// TIA Portal project "传感器对中" (V15.1)

(* hardware
DEVICE "S7-1200 station_1"  S7-1200 Station
   slot 0: "Rack_0"  S7-1200 Rack  Rack  V1.0
   slot 1: "280PLC"  CPU 1214C DC/DC/DC  6ES7 214-1AG40-0XB0  V4.2
   slot 2: "DI 16x24VDC/DQ 16xRelay_1"  SM 1223 DI16/DQ16 x relay  6ES7 223-1PL32-0XB0  V2.0
   slot 3: "DI 16/DQ 16x24VDC_1"  6ES7 223-1BL32-0XB0  V2.0
   slot 4: "DI 8x24VDC_1"  6ES7 221-1BF32-0XB0  V2.0
   slot 5: "AI 4x13BIT_1"  6ES7 231-4HD32-0XB0  V2.0
DEVICE "GSD device_1"  GSD.Device.PN
   slot 0: "机架"  Rack  V1.0
   slot 0: "1-sr-qd1"  SINAMICS V90 PN V1.0  6SL3 210-5Fxxx-xxFx  V1.00
      slot 0: "SINAMICS V90 PN V1.0"  SINAMICS V90 PN V1.0
      slot 1: "PN-IO"  PN-IO
         slot 1: "端口1"  Port 1
         slot 2: "端口2"  Port 2
      slot 1: "驱动_1"  Drive
         slot 0: "模块访问点"  Module Access Point
         slot 1: "没有 PROFIsafe"  without PROFIsafe
   slot 2: "标准报文3, PZD-5/9"  Standard telegram 3, PZD-5/9
DEVICE "GSD device_2"  GSD.Device.PN
   slot 0: "机架"  Rack  V1.0
   slot 0: "2-sr-qd2"  SINAMICS V90 PN V1.0  6SL3 210-5Fxxx-xxFx  V1.00
      slot 0: "SINAMICS V90 PN V1.0"  SINAMICS V90 PN V1.0
      slot 1: "PN-IO"  PN-IO
         slot 1: "端口1"  Port 1
         slot 2: "端口2"  Port 2
      slot 1: "驱动_1"  Drive
         slot 0: "模块访问点"  Module Access Point
         slot 1: "没有 PROFIsafe"  without PROFIsafe
   slot 2: "标准报文3, PZD-5/9"  Standard telegram 3, PZD-5/9
DEVICE "GSD device_4"  GSD.Device.PN
   slot 0: "机架"  Rack  V1.0
   slot 0: "4-sr-yz2"  SINAMICS V90 PN V1.0  6SL3 210-5Fxxx-xxFx  V1.00
      slot 0: "SINAMICS V90 PN V1.0"  SINAMICS V90 PN V1.0
      slot 1: "PN-IO"  PN-IO
         slot 1: "端口1"  Port 1
         slot 2: "端口2"  Port 2
      slot 1: "驱动_1"  Drive
         slot 0: "模块访问点"  Module Access Point
         slot 1: "没有 PROFIsafe"  without PROFIsafe
   slot 2: "标准报文3, PZD-5/9"  Standard telegram 3, PZD-5/9
DEVICE "GSD device_3"  GSD.Device.PN
   slot 0: "机架"  Rack  V1.0
   slot 0: "3-sr-yz1"  SINAMICS V90 PN V1.0  6SL3 210-5Fxxx-xxFx  V1.00
      slot 0: "SINAMICS V90 PN V1.0"  SINAMICS V90 PN V1.0
      slot 1: "PN-IO"  PN-IO
         slot 1: "端口1"  Port 1
         slot 2: "端口2"  Port 2
      slot 1: "驱动_1"  Drive
         slot 0: "模块访问点"  Module Access Point
         slot 1: "没有 PROFIsafe"  without PROFIsafe
   slot 2: "标准报文3, PZD-5/9"  Standard telegram 3, PZD-5/9
*)

// ===== PLC "280PLC"  CPU 1214C DC/DC/DC =====

VAR_GLOBAL   // PLC tag table "默认变量表"
   "角度编码器1A" AT %I0.0 : Bool;
   "角度编码器1B" AT %I0.1 : Bool;
   "角度编码器1Z" AT %I0.3 : Bool;
   "角度编码器2A" AT %I0.4 : Bool;
   "角度编码器2B" AT %I0.5 : Bool;
   "角度编码器2Z" AT %I0.7 : Bool;
   "工位1在位" AT %I1.4 : Bool;
   "工位2在位" AT %I1.5 : Bool;
   "工位1卡盘顶升进到位" AT %I2.0 : Bool;
   "工位1卡盘顶升退到位" AT %I2.1 : Bool;
   "产品扶持气缸1进到位" AT %I2.2 : Bool;
   "产品扶持气缸1退到位" AT %I2.3 : Bool;
   "输出轴夹紧气缸1进到位" AT %I5.4 : Bool;
   "输出轴夹紧气缸1退到位" AT %I5.5 : Bool;
   "输出轴花键移载气缸1进到位" AT %I2.6 : Bool;
   "输出轴花键移载气缸1退到位" AT %I2.7 : Bool;
   "输入轴夹紧气动卡盘2进到位" AT %I3.0 : Bool;
   "输入轴夹紧气动卡盘2退到位" AT %I3.1 : Bool;
   "产品扶持气缸2进到位" AT %I3.2 : Bool;
   "产品扶持气缸2退到位" AT %I3.3 : Bool;
   "输出轴夹紧气缸2进到位" AT %I5.6 : Bool;
   "输出轴夹紧气缸2退到位" AT %I5.7 : Bool;
   "输出轴花键移载气缸2进到位" AT %I3.6 : Bool;
   "输出轴花键移载气缸2退到位" AT %I3.7 : Bool;
   "工位2启动" AT %I4.0 : Bool;
   "复位按钮" AT %I4.1 : Bool;
   "工位1启动" AT %I4.2 : Bool;
   "安全光栅" AT %I4.3 : Bool;
   "安全继电器急停" AT %I4.4 : Bool;
   "安全门开关" AT %I4.5 : Bool;
   "急停按钮" AT %I4.6 : Bool;
   "气源不足指示" AT %I4.7 : Bool;
   "报警1" AT %I5.0 : Bool;
   "报警2" AT %I5.1 : Bool;
   "报警3" AT %I5.2 : Bool;
   "报警4" AT %I5.3 : Bool;
   "扭矩传感器1" AT %IW144 : Int;
   "扭矩传感器2" AT %IW146 : Int;
   "输入轴移载伺服-1_归位开关" AT %I1.0 : Bool;
   "输入轴移载伺服-2_归位开关" AT %I1.3 : Bool;
   "输入轴驱动伺服-1_Drive_IN" AT %I68.0 : "PD_TEL3_IN";
   "输入轴驱动伺服-2_Drive_IN" AT %I104.0 : "PD_TEL3_IN";
   "输入轴驱动伺服-2_Drive_IN(1)" AT %I86.0 : "PD_TEL3_IN";
   "输入轴移载伺服-1_Drive_IN" AT %I122.0 : "PD_TEL3_IN";
   "输入轴移载伺服-1_LowHwLimitSwitch" AT %I0.6 : Bool;
   "输入轴移载伺服-1_HighHwLimitSwitch" AT %I0.2 : Bool;
   "输入轴移载伺服-2_LowHwLimitSwitch" AT %I1.2 : Bool;
   "输入轴移载伺服-2_HighHwLimitSwitch" AT %I1.1 : Bool;
   "编码器计数1" AT %ID1000 : DInt;
   "编码器计数2" AT %ID1004 : DInt;
   "Tag_8" AT %IW1000 : Hw_Hsc;
   "输入轴驱动伺服-1_归位开关" AT %I3.4 : Bool;
   "输入轴驱动伺服-2_归位开关" AT %I3.5 : Bool;
   "工位2卡盘顶升进到位" AT %I2.4 : Bool;
   "工位2卡盘顶升退到位" AT %I2.5 : Bool;
   "复位1" AT %Q0.0 : Bool;
   "复位2" AT %Q0.1 : Bool;
   "复位3" AT %Q0.2 : Bool;
   "复位4" AT %Q0.3 : Bool;
   "三色灯-红" AT %Q0.4 : Bool;
   "三色灯-黄" AT %Q0.5 : Bool;
   "三色灯-绿" AT %Q0.6 : Bool;
   "蜂鸣器" AT %Q0.7 : Bool;
   "输入轴夹紧气动卡盘1进" AT %Q2.0 : Bool;
   "输入轴夹紧气动卡盘1退" AT %Q2.1 : Bool;
   "产品扶持气缸1进" AT %Q2.2 : Bool;
   "产品扶持气缸1退" AT %Q2.3 : Bool;
   "输出轴夹紧气缸1进" AT %Q2.4 : Bool;
   "输出轴夹紧气缸1退" AT %Q2.5 : Bool;
   "输出轴花键移载气缸1进" AT %Q2.6 : Bool;
   "输出轴花键移载气缸1退" AT %Q2.7 : Bool;
   "输入轴夹紧气动卡盘2进" AT %Q3.0 : Bool;
   "输入轴夹紧气动卡盘2退" AT %Q3.1 : Bool;
   "产品扶持气缸2进" AT %Q3.2 : Bool;
   "产品扶持气缸2退" AT %Q3.3 : Bool;
   "输出轴夹紧气缸2进" AT %Q3.4 : Bool;
   "输出轴夹紧气缸2退" AT %Q3.5 : Bool;
   "输出轴花键移载气缸2进" AT %Q3.6 : Bool;
   "输出轴花键移载气缸2退" AT %Q3.7 : Bool;
   "工位1两色灯-红" AT %Q4.0 : Bool;
   "工位1两色灯-绿" AT %Q4.1 : Bool;
   "工位2两色灯-红" AT %Q4.2 : Bool;
   "工位2两色灯-绿" AT %Q4.3 : Bool;
   "总气阀" AT %Q4.4 : Bool;
   "工位1采集切换" AT %Q4.6 : Bool;   // True:PGI采集False:板卡采集
   "输入轴驱动伺服-1_Drive_OUT" AT %Q64.0 : "PD_TEL3_OUT";
   "输入轴驱动伺服-2_Drive_OUT" AT %Q84.0 : "PD_TEL3_OUT";
   "输入轴驱动伺服-2_Drive_OUT(1)" AT %Q74.0 : "PD_TEL3_OUT";
   "输入轴移载伺服-1_Drive_OUT" AT %Q94.0 : "PD_TEL3_OUT";
   "工位2采集切换" AT %Q4.5 : Bool;   // True:PGI采集False:板卡采集
   "工位1卡盘顶升进" AT %Q5.0 : Bool;
   "工位1卡盘顶升退" AT %Q5.1 : Bool;
   "工位2卡盘顶升进" AT %Q5.2 : Bool;
   "工位2卡盘顶升退" AT %Q5.3 : Bool;
   "System_Byte" AT %MB1 : Byte;
   "FirstScan" AT %M1.0 : Bool;
   "DiagStatusUpdate" AT %M1.1 : Bool;
   "AlwaysTRUE" AT %M1.2 : Bool;
   "AlwaysFALSE" AT %M1.3 : Bool;
   "Clock_Byte" AT %MB0 : Byte;
   "Clock_10Hz" AT %M0.0 : Bool;
   "Clock_5Hz" AT %M0.1 : Bool;
   "Clock_2.5Hz" AT %M0.2 : Bool;
   "Clock_2Hz" AT %M0.3 : Bool;
   "Clock_1.25Hz" AT %M0.4 : Bool;
   "Clock_1Hz" AT %M0.5 : Bool;
   "Clock_0.625Hz" AT %M0.6 : Bool;
   "Clock_0.5Hz" AT %M0.7 : Bool;
   "单工位1" AT %M100.0 : Bool;
   "单工位2" AT %M100.1 : Bool;
   "程序停止" AT %M100.3 : Bool;
   "光栅启用" AT %M100.2 : Bool;
   "急停拍下故障" AT %M110.0 : Bool;
   "气源不足故障" AT %M110.1 : Bool;
   "安全门打开故障" AT %M110.2 : Bool;
   "光栅触碰故障" AT %M110.3 : Bool;
   "输入轴夹紧气动卡盘1进故障" AT %M110.4 : Bool;
   "输入轴夹紧气动卡盘1退故障" AT %M110.5 : Bool;
   "产品扶持气缸1进故障" AT %M110.6 : Bool;
   "产品扶持气缸1退故障" AT %M110.7 : Bool;
   "输出轴夹紧气缸1进故障" AT %M111.0 : Bool;
   "输出轴夹紧气缸1退故障" AT %M111.1 : Bool;
   "输出轴花键移载气缸1进故障" AT %M111.2 : Bool;
   "输出轴花键移载气缸1退故障" AT %M111.3 : Bool;
   "输入轴夹紧气动卡盘2进故障" AT %M111.4 : Bool;
   "输入轴夹紧气动卡盘2退故障" AT %M111.5 : Bool;
   "产品扶持气缸2进故障" AT %M111.6 : Bool;
   "产品扶持气缸2退故障" AT %M111.7 : Bool;
   "输出轴夹紧气缸2进故障" AT %M112.0 : Bool;
   "输出轴夹紧气缸2退故障" AT %M112.1 : Bool;
   "输出轴花键移载气缸2进故障" AT %M112.2 : Bool;
   "输出轴花键移载气缸2退故障" AT %M112.3 : Bool;
   "输入轴移载伺服1退到位故障" AT %M120.0 : Bool;
   "输入轴移载伺服1进到位故障" AT %M120.1 : Bool;
   "输入轴移载伺服2退到位故障" AT %M120.2 : Bool;
   "输入轴移载伺服2进到位故障" AT %M120.3 : Bool;
   "输入轴驱动伺服-1故障" AT %M130.0 : Bool;
   "输入轴驱动伺服-2故障" AT %M130.1 : Bool;
   "输入轴移载伺服-1故障" AT %M130.2 : Bool;
   "输入轴移载伺服-2故障" AT %M130.3 : Bool;
   "复位启动" AT %M100.4 : Bool;
   "复位完成" AT %M100.5 : Bool;
   "Tag_4" AT %M3.3 : Bool;
   "复位停止" AT %M100.6 : Bool;
   "Tag_5" AT %M3.4 : Bool;
   "复位电机" AT %M100.7 : Bool;
   "中断power" AT %M101.0 : Bool;
   "Tag_6" AT %M3.5 : Bool;
   "复位高速1" AT %M101.1 : Bool;
   "复位高速2" AT %M101.2 : Bool;
   "系统报警" AT %MW110 : Int;
   "电机报警" AT %MW112 : Int;
   "气缸报警" AT %MW114 : Int;
   "测试1" AT %M200.0 : Bool;
   "复位" AT %M101.3 : Bool;
   "Tag_9" AT %M4.0 : Bool;
   "Tag_10" AT %M4.1 : Bool;
   "Tag_11" AT %M4.2 : Bool;
   "测试2" AT %M200.1 : Bool;
   "显示1" AT %MD210 : Real;
   "显示2" AT %MD214 : Real;
   "测试结束1" AT %M200.2 : Bool;
   "测试结束2" AT %M200.3 : Bool;
   "Tag_7" AT %M4.3 : Bool;
   "Tag_12" AT %M4.4 : Bool;
   "Tag_1" AT %MW2000 : Word;
END_VAR

DATA_BLOCK "Auto2_DB"   // DB1
{ S7_Optimized_Access := 'TRUE' }
VERSION : 0.1
// stored: InstanceOfName Auto2
"Auto2"
BEGIN
END_DATA_BLOCK

DATA_BLOCK "SERVER_DB"   // DB2
{ S7_Optimized_Access := 'FALSE' }
VERSION : 0.1
   VAR
      设备状态 : Int;
      错误代码 : Int;
      工位1状态 : Int;
      工位2状态 : Int;
      传感器 : Array[0..7] of Real;
      工位一驱动伺服参数 : Array[0..3] of Real;
      工位二驱动伺服参数 : Array[0..3] of Real;
      工位一移载伺服手动参数 : Array[0..3] of Real;
      工位一移载伺服自动参数 : Array[0..3] of Real;
      工位二移载伺服手动参数 : Array[0..3] of Real;
      工位二移载伺服自动参数 : Array[0..3] of Real;
      工位一扭矩传感器参数 : Array[0..4] of Real;
      工位二扭矩传感器参数 : Array[0..4] of Real;
      复检参数 : Array[0..5] of Real;
      动态优化参数 : Array[0..5] of Real;
      合格状态 : Int;
      合格状态2 : Int;
      工位一暂停 : Int;
      工位二暂停 : Int;
   END_VAR
BEGIN
   工位一扭矩传感器参数[0] := 0.0;   // 量程下限
   工位一扭矩传感器参数[1] := 50.0;   // 量程上限
   工位二扭矩传感器参数[0] := 0.0;   // 量程下限
   工位二扭矩传感器参数[1] := 50.0;   // 量程上限
   工位一驱动伺服参数[0] := 15.0;   // 状态
   工位二驱动伺服参数[0] := 15.0;   // 状态
   工位一扭矩传感器参数[3] := 0.0;   // 正向偏移
   // 传感器[0] : 输入轴驱动伺服-1
   // 传感器[1] : 输入轴驱动伺服-2
   // 传感器[2] : 输入轴移载伺服-1
   // 传感器[3] : 输入轴移载伺服-2
   // 工位一驱动伺服参数[1] : 速度
   // 工位一驱动伺服参数[2] : 相对位置
   // 工位一驱动伺服参数[3] : 绝对位置
   // 工位一扭矩传感器参数[2] : 原始值
   // 工位一扭矩传感器参数[4] : 逆向偏移
   // 工位二扭矩传感器参数[2] : 原始值
   // 工位二扭矩传感器参数[3] : 正向偏移
   // 工位二扭矩传感器参数[4] : 逆向偏移
   // 传感器[4] : 编码器1
   // 传感器[5] : 编码器2
   // 工位二驱动伺服参数[1] : 速度
   // 工位二驱动伺服参数[2] : 相对位置
   // 工位二驱动伺服参数[3] : 绝对位置
   // 工位一移载伺服手动参数[0] : 状态
   // 工位一移载伺服手动参数[1] : 速度
   // 工位一移载伺服手动参数[2] : 相对位置
   // 工位一移载伺服手动参数[3] : 绝对位置
   // 工位二移载伺服手动参数[0] : 状态
   // 工位二移载伺服手动参数[1] : 速度
   // 工位二移载伺服手动参数[2] : 相对位置
   // 工位二移载伺服手动参数[3] : 绝对位置
   // 工位一移载伺服自动参数[0] : 接近位置
   // 工位一移载伺服自动参数[1] : 接近速度
   // 工位一移载伺服自动参数[2] : 最终位置
   // 工位一移载伺服自动参数[3] : 最终速度
   // 工位二移载伺服自动参数[0] : 接近位置
   // 工位二移载伺服自动参数[1] : 接近速度
   // 工位二移载伺服自动参数[2] : 最终位置
   // 工位二移载伺服自动参数[3] : 最终速度
   // 传感器[6] : 工位一扭矩
   // 传感器[7] : 工位二扭矩
   // 复检参数[0] : 复检速度
   // 复检参数[1] : 复检扭矩
   // 复检参数[2] : 工位一卡盘夹紧位置
   // 复检参数[3] : 工位一卡盘松开位置
   // 复检参数[4] : 工位二卡盘夹紧位置
   // 复检参数[5] : 工位二卡盘松开位置
   // 动态优化参数[0] : 动态优化速度
   // 动态优化参数[1] : 动态优化角度
   // 动态优化参数[2] : 动态优化复测速度
   // 动态优化参数[3] : 对称性
END_DATA_BLOCK

DATA_BLOCK "Auto1_DB"   // DB3
{ S7_Optimized_Access := 'TRUE' }
VERSION : 0.1
// stored: InstanceOfName Auto1
"Auto1"
BEGIN
END_DATA_BLOCK

DATA_BLOCK "All_Servo_DB"   // DB16
{ S7_Optimized_Access := 'TRUE' }
VERSION : 0.1
// stored: InstanceOfName All_Servo
"All_Servo"
BEGIN
END_DATA_BLOCK

DATA_BLOCK "Reset_DB"   // DB20
{ S7_Optimized_Access := 'TRUE' }
VERSION : 0.1
// stored: InstanceOfName Reset
"Reset"
BEGIN
END_DATA_BLOCK

DATA_BLOCK "Alarm_DB"   // DB23
{ S7_Optimized_Access := 'TRUE' }
VERSION : 0.1
// stored: InstanceOfName Alarm
"Alarm"
BEGIN
END_DATA_BLOCK

// folder: System blocks/Program resources

DATA_BLOCK "IEC_Timer_0_DB"   // DB24
{ S7_Optimized_Access := 'TRUE' }
AUTHOR : Simatic
FAMILY : IEC
NAME : IEC_TMR
VERSION : 1.0
// stored: InstanceOfName IEC_TIMER
"IEC_TIMER"
BEGIN
END_DATA_BLOCK

// folder: (top level)

DATA_BLOCK "输入轴驱动伺服-1"   // DB4, Motion_DB
{ S7_Optimized_Access := 'TRUE' }
AUTHOR : SIMATIC
FAMILY : BasicMC
NAME : TO_PosAx
VERSION : 6.0
// stored: InstanceOfName TO_PositioningAxis
"TO_PositioningAxis"
BEGIN
   // Axis.HomingReferencePointSwitch_AddressCU = %I3.4
   // Axis.LengthUnit.LastDistance = 1005
   // Axis.Encoder.TelegramAddressOutCU = %Q64.0
   // Axis.Encoder.TelegramAddressInCU = %I68.0
   // Axis.Encoder.OutputAddress = 64
   // Axis.Encoder.InputAddress = 68
   // Axis.Encoder.DoNameCU = 1-sr-qd1.驱动_1_编码器1
   // Axis.Drive.OutputAddress = 64
   // Axis.Drive.InputAddress = 68
   // Axis.Drive.TelegramAddressOutCU = %Q64.0
   // Axis.Drive.TelegramAddressInCU = %I68.0
   // Axis.Drive.DoNameCU = 1-sr-qd1.驱动_1
   // Axis.Drive.TelegramType = 2
   // Axis.LengthUnitNormalized.Distance = 1005
   // Axis.Encoder.SelectedHscIndexCU = -1
   // Axis.Encoder.DbTypeCU = Classic
   // Axis.Drive.DbTypeCU = Classic
END_DATA_BLOCK

DATA_BLOCK "输入轴移载伺服-1"   // DB5, Motion_DB
{ S7_Optimized_Access := 'TRUE' }
AUTHOR : SIMATIC
FAMILY : BasicMC
NAME : TO_PosAx
VERSION : 6.0
// stored: InstanceOfName TO_PositioningAxis
"TO_PositioningAxis"
BEGIN
   // Axis.PositionLimitsMax_AddressCU = %I0.2
   // Axis.PositionLimitsMin_AddressCU = %I0.6
   // Axis.HomingReferencePointSwitch_AddressCU = %I1.0
   // Axis.Encoder.TelegramAddressOutCU = %Q94.0
   // Axis.Encoder.TelegramAddressInCU = %I122.0
   // Axis.Encoder.OutputAddress = 94
   // Axis.Encoder.InputAddress = 122
   // Axis.Encoder.DoNameCU = 3-sr-yz1.驱动_1_编码器1
   // Axis.Drive.OutputAddress = 94
   // Axis.Drive.InputAddress = 122
   // Axis.Drive.TelegramAddressOutCU = %Q94.0
   // Axis.Drive.TelegramAddressInCU = %I122.0
   // Axis.Drive.TelegramType = 2
   // Axis.Drive.DoNameCU = 3-sr-yz1.驱动_1
   // Axis.LengthUnitNormalized.Distance = 1013
   // Axis.Encoder.SelectedHscIndexCU = -1
   // Axis.Encoder.DbTypeCU = Classic
   // Axis.Drive.DbTypeCU = Classic
END_DATA_BLOCK

DATA_BLOCK "输入轴驱动伺服-2"   // DB6, Motion_DB
{ S7_Optimized_Access := 'TRUE' }
AUTHOR : SIMATIC
FAMILY : BasicMC
NAME : TO_PosAx
VERSION : 6.0
// stored: InstanceOfName TO_PositioningAxis
"TO_PositioningAxis"
BEGIN
   // Axis.HomingReferencePointSwitch_AddressCU = %I3.5
   // Axis.LengthUnit.LastDistance = 1005
   // Axis.Encoder.TelegramAddressOutCU = %Q74.0
   // Axis.Encoder.TelegramAddressInCU = %I86.0
   // Axis.Encoder.OutputAddress = 74
   // Axis.Encoder.InputAddress = 86
   // Axis.Encoder.DoNameCU = 2-sr-qd2.驱动_1_编码器1
   // Axis.Drive.OutputAddress = 74
   // Axis.Drive.InputAddress = 86
   // Axis.Drive.TelegramAddressOutCU = %Q74.0
   // Axis.Drive.TelegramAddressInCU = %I86.0
   // Axis.Drive.TelegramType = 2
   // Axis.Drive.DoNameCU = 2-sr-qd2.驱动_1
   // Axis.LengthUnitNormalized.Distance = 1005
   // Axis.Encoder.SelectedHscIndexCU = -1
   // Axis.Encoder.DbTypeCU = Classic
   // Axis.Drive.DbTypeCU = Classic
END_DATA_BLOCK

DATA_BLOCK "输入轴移载伺服-2"   // DB7, Motion_DB
{ S7_Optimized_Access := 'TRUE' }
AUTHOR : SIMATIC
FAMILY : BasicMC
NAME : TO_PosAx
VERSION : 6.0
// stored: InstanceOfName TO_PositioningAxis
"TO_PositioningAxis"
BEGIN
   // Axis.PositionLimitsMax_AddressCU = %I1.1
   // Axis.PositionLimitsMin_AddressCU = %I1.2
   // Axis.HomingReferencePointSwitch_AddressCU = %I1.3
   // Axis.Encoder.TelegramAddressOutCU = %Q84.0
   // Axis.Encoder.TelegramAddressInCU = %I104.0
   // Axis.Encoder.OutputAddress = 84
   // Axis.Encoder.InputAddress = 104
   // Axis.Encoder.DoNameCU = 4-sr-yz2.驱动_1_编码器1
   // Axis.Drive.OutputAddress = 84
   // Axis.Drive.InputAddress = 104
   // Axis.Drive.TelegramAddressOutCU = %Q84.0
   // Axis.Drive.TelegramAddressInCU = %I104.0
   // Axis.Drive.TelegramType = 2
   // Axis.Drive.DoNameCU = 4-sr-yz2.驱动_1
   // Axis.LengthUnitNormalized.Distance = 1013
   // Axis.Encoder.SelectedHscIndexCU = -1
   // Axis.Encoder.DbTypeCU = Classic
   // Axis.Drive.DbTypeCU = Classic
END_DATA_BLOCK

FUNCTION_BLOCK "Servo"   // FB1, LAD
{ S7_Optimized_Access := 'TRUE' }
VERSION : 0.1
   VAR_INPUT
      Axis : TO_PositioningAxis;
      SON : Bool;
      Reset : Bool;
      Mode : Int;
      MoveHome : Bool;
      Halt : Bool;
      Position : Real;
      Velocity : Real;
      JogForword : Bool;
      JogBackword : Bool;
      MoveAbsolute : Bool;
      MoveRelative : Bool;
   END_VAR
   VAR
      MC_Power_Instance : MC_Power;
      MC_Reset_Instance : MC_Reset;
      MC_Halt_Instance : MC_Halt;
      MC_MoveAbsolute_Instance : MC_MoveAbsolute;
      MC_MoveRelative_Instance : MC_MoveRelative;
      MC_MoveJog_Instance : MC_MoveJog;
      MC_Home_Instance : MC_Home;
   END_VAR
BEGIN

REGION Network 1
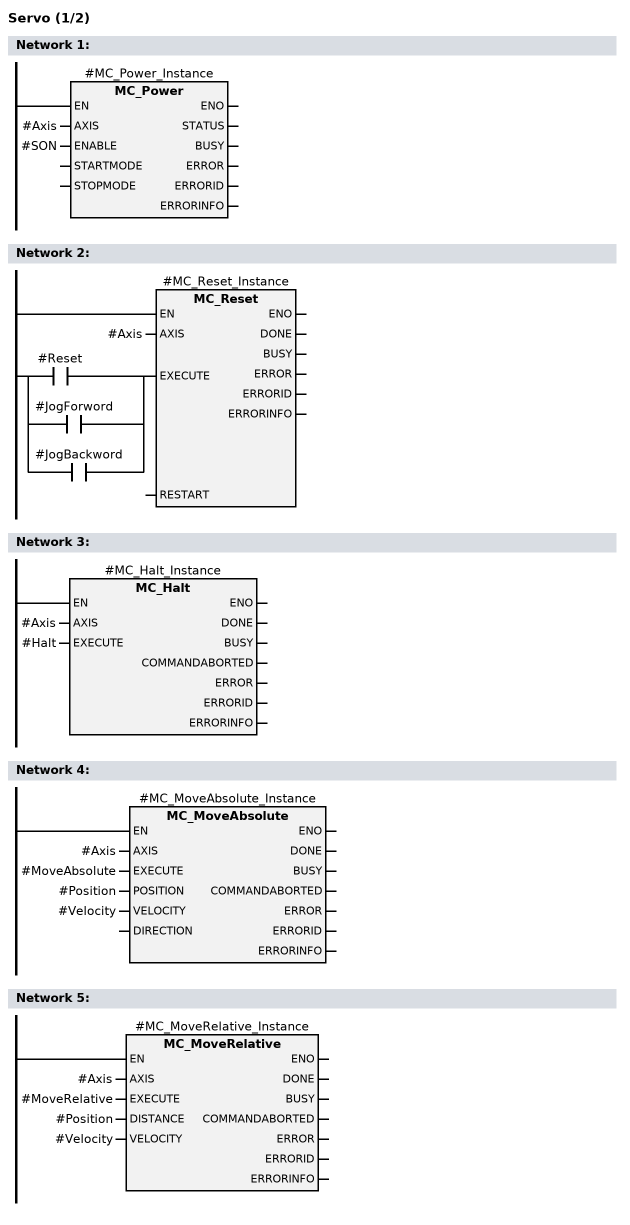
   #MC_Power_Instance(Axis := #Axis, Enable := #SON);   // MC_Power
END_REGION

REGION Network 2
   #MC_Reset_Instance(Axis := #Axis, Execute := #Reset OR #JogForword OR #JogBackword);   // MC_Reset
END_REGION

REGION Network 3
   #MC_Halt_Instance(Axis := #Axis, Execute := #Halt);   // MC_Halt
END_REGION

REGION Network 4
   #MC_MoveAbsolute_Instance(Axis := #Axis,   // MC_MoveAbsolute
                           Execute := #MoveAbsolute,
                           Position := #Position,
                           Velocity := #Velocity);
END_REGION

REGION Network 5
   #MC_MoveRelative_Instance(Axis := #Axis,   // MC_MoveRelative
                           Execute := #MoveRelative,
                           Distance := #Position,
                           Velocity := #Velocity);
END_REGION

REGION Network 6
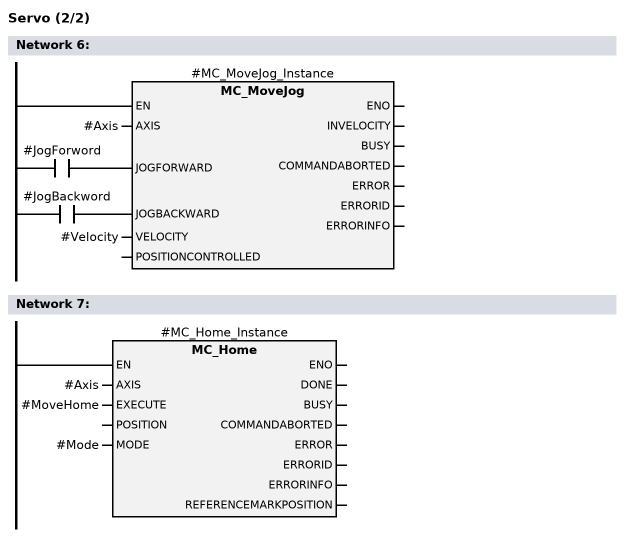
   #MC_MoveJog_Instance(Axis := #Axis,   // MC_MoveJog
                        JogForward := #JogForword,
                        JogBackward := #JogBackword,
                        Velocity := #Velocity);
END_REGION

REGION Network 7
   #MC_Home_Instance(Axis := #Axis, Execute := #MoveHome, Mode := #Mode);   // MC_Home
END_REGION
END_FUNCTION_BLOCK

FUNCTION_BLOCK "All_Servo"   // FB2, LAD
TITLE = 手动调试电机
{ S7_Optimized_Access := 'TRUE' }
VERSION : 0.1
   VAR
      Servo_Instance : "Servo";
      Servo_Instance_1 : "Servo";
      Servo_Instance_2 : "Servo";
      Servo_Instance_3 : "Servo";
   END_VAR
BEGIN

REGION Network 1: 手动输入轴驱动伺服-1
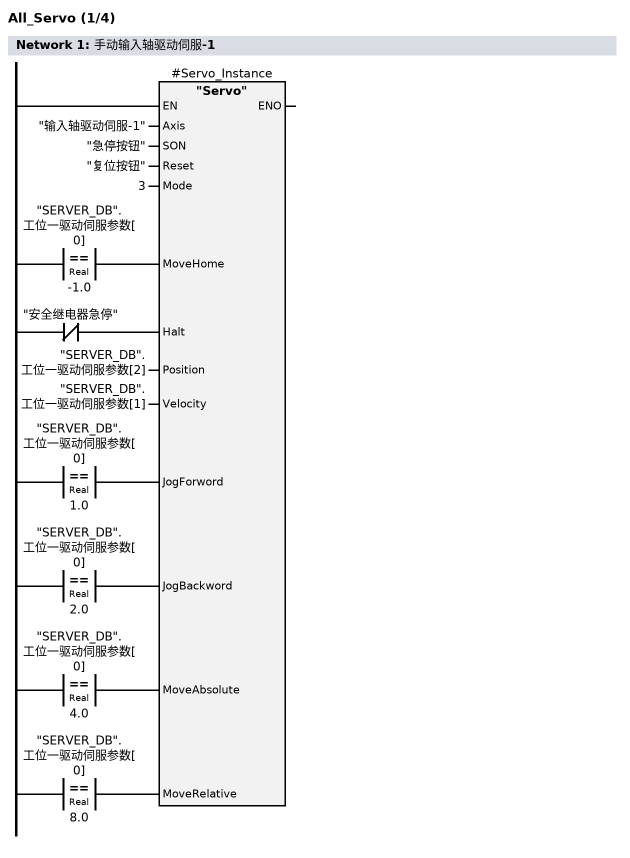
   RUNG wire#powerrail
      #Servo_Instance(MoveHome := wire#w1, Halt := wire#w2, JogForword := wire#w3, JogBackword := wire#w4, MoveAbsolute := wire#w5, MoveRelative := wire#w6, Axis := "输入轴驱动伺服-1", SON := "急停按钮", Reset := "复位按钮", Mode := 3, Position := "SERVER_DB".工位一驱动伺服参数[2], Velocity := "SERVER_DB".工位一驱动伺服参数[1])
   END_RUNG
   RUNG wire#powerrail
      { S7_Templates := "SrcType := Real" } EQ_Contact(in1 := "SERVER_DB".工位一驱动伺服参数[0], in2 := -1.0)
   END_RUNG wire#w1
   RUNG wire#powerrail
      I_Contact( "安全继电器急停" )
   END_RUNG wire#w2
   RUNG wire#powerrail
      { S7_Templates := "SrcType := Real" } EQ_Contact(in1 := "SERVER_DB".工位一驱动伺服参数[0], in2 := 1.0)
   END_RUNG wire#w3
   RUNG wire#powerrail
      { S7_Templates := "SrcType := Real" } EQ_Contact(in1 := "SERVER_DB".工位一驱动伺服参数[0], in2 := 2.0)
   END_RUNG wire#w4
   RUNG wire#powerrail
      { S7_Templates := "SrcType := Real" } EQ_Contact(in1 := "SERVER_DB".工位一驱动伺服参数[0], in2 := 4.0)
   END_RUNG wire#w5
   RUNG wire#powerrail
      { S7_Templates := "SrcType := Real" } EQ_Contact(in1 := "SERVER_DB".工位一驱动伺服参数[0], in2 := 8.0)
   END_RUNG wire#w6
   // the same network as SCL:
   #Servo_Instance(Axis := "输入轴驱动伺服-1",   // "Servo"
                   SON := "急停按钮",
                   Reset := "复位按钮",
                   Mode := 3,
                   MoveHome := "SERVER_DB".工位一驱动伺服参数[0] = (-1.0),
                   Halt := NOT "安全继电器急停",
                   Position := "SERVER_DB".工位一驱动伺服参数[2],
                   Velocity := "SERVER_DB".工位一驱动伺服参数[1],
                   JogForword := "SERVER_DB".工位一驱动伺服参数[0] = 1.0,
                   JogBackword := "SERVER_DB".工位一驱动伺服参数[0] = 2.0,
                   MoveAbsolute := "SERVER_DB".工位一驱动伺服参数[0] = 4.0,
                   MoveRelative := "SERVER_DB".工位一驱动伺服参数[0] = 8.0);
END_REGION

REGION Network 2: 手动输入轴驱动伺服-2
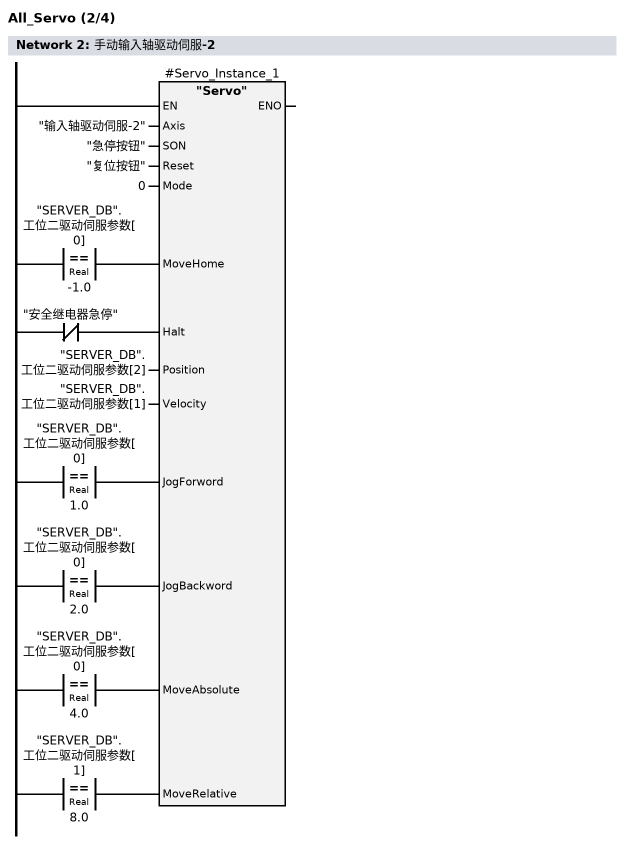
   RUNG wire#powerrail
      #Servo_Instance_1(MoveHome := wire#w1, Halt := wire#w2, JogForword := wire#w3, JogBackword := wire#w4, MoveAbsolute := wire#w5, MoveRelative := wire#w6, Axis := "输入轴驱动伺服-2", SON := "急停按钮", Reset := "复位按钮", Mode := 0, Position := "SERVER_DB".工位二驱动伺服参数[2], Velocity := "SERVER_DB".工位二驱动伺服参数[1])
   END_RUNG
   RUNG wire#powerrail
      { S7_Templates := "SrcType := Real" } EQ_Contact(in1 := "SERVER_DB".工位二驱动伺服参数[0], in2 := -1.0)
   END_RUNG wire#w1
   RUNG wire#powerrail
      I_Contact( "安全继电器急停" )
   END_RUNG wire#w2
   RUNG wire#powerrail
      { S7_Templates := "SrcType := Real" } EQ_Contact(in1 := "SERVER_DB".工位二驱动伺服参数[0], in2 := 1.0)
   END_RUNG wire#w3
   RUNG wire#powerrail
      { S7_Templates := "SrcType := Real" } EQ_Contact(in1 := "SERVER_DB".工位二驱动伺服参数[0], in2 := 2.0)
   END_RUNG wire#w4
   RUNG wire#powerrail
      { S7_Templates := "SrcType := Real" } EQ_Contact(in1 := "SERVER_DB".工位二驱动伺服参数[0], in2 := 4.0)
   END_RUNG wire#w5
   RUNG wire#powerrail
      { S7_Templates := "SrcType := Real" } EQ_Contact(in1 := "SERVER_DB".工位二驱动伺服参数[1], in2 := 8.0)
   END_RUNG wire#w6
   // the same network as SCL:
   #Servo_Instance_1(Axis := "输入轴驱动伺服-2",   // "Servo"
                     SON := "急停按钮",
                     Reset := "复位按钮",
                     Mode := 0,
                     MoveHome := "SERVER_DB".工位二驱动伺服参数[0] = (-1.0),
                     Halt := NOT "安全继电器急停",
                     Position := "SERVER_DB".工位二驱动伺服参数[2],
                     Velocity := "SERVER_DB".工位二驱动伺服参数[1],
                     JogForword := "SERVER_DB".工位二驱动伺服参数[0] = 1.0,
                     JogBackword := "SERVER_DB".工位二驱动伺服参数[0] = 2.0,
                     MoveAbsolute := "SERVER_DB".工位二驱动伺服参数[0] = 4.0,
                     MoveRelative := "SERVER_DB".工位二驱动伺服参数[1] = 8.0);
END_REGION

REGION Network 3: 手动输入轴移载伺服-1
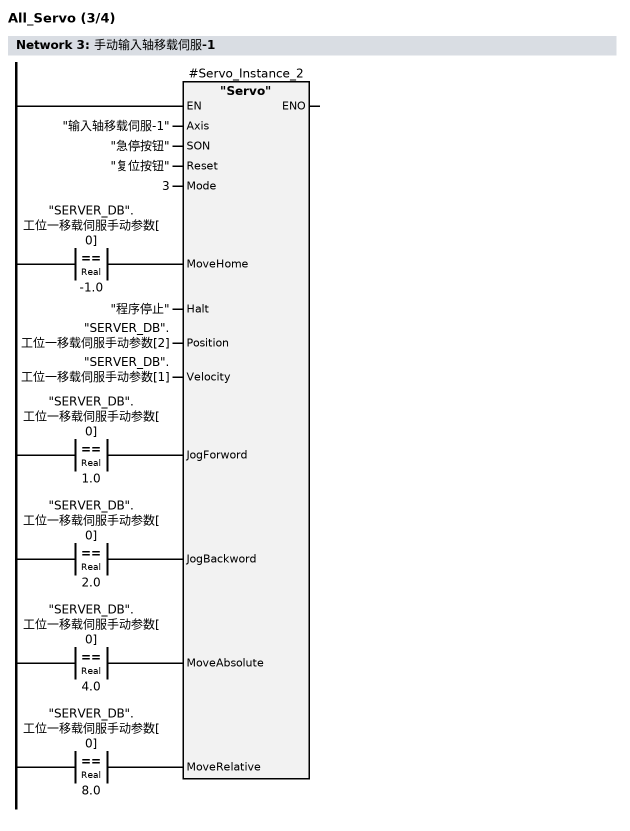
   RUNG wire#powerrail
      #Servo_Instance_2(MoveHome := wire#w1, JogForword := wire#w2, JogBackword := wire#w3, MoveAbsolute := wire#w4, MoveRelative := wire#w5, Axis := "输入轴移载伺服-1", SON := "急停按钮", Reset := "复位按钮", Mode := 3, Halt := "程序停止", Position := "SERVER_DB".工位一移载伺服手动参数[2], Velocity := "SERVER_DB".工位一移载伺服手动参数[1])
   END_RUNG
   RUNG wire#powerrail
      { S7_Templates := "SrcType := Real" } EQ_Contact(in1 := "SERVER_DB".工位一移载伺服手动参数[0], in2 := -1.0)
   END_RUNG wire#w1
   RUNG wire#powerrail
      { S7_Templates := "SrcType := Real" } EQ_Contact(in1 := "SERVER_DB".工位一移载伺服手动参数[0], in2 := 1.0)
   END_RUNG wire#w2
   RUNG wire#powerrail
      { S7_Templates := "SrcType := Real" } EQ_Contact(in1 := "SERVER_DB".工位一移载伺服手动参数[0], in2 := 2.0)
   END_RUNG wire#w3
   RUNG wire#powerrail
      { S7_Templates := "SrcType := Real" } EQ_Contact(in1 := "SERVER_DB".工位一移载伺服手动参数[0], in2 := 4.0)
   END_RUNG wire#w4
   RUNG wire#powerrail
      { S7_Templates := "SrcType := Real" } EQ_Contact(in1 := "SERVER_DB".工位一移载伺服手动参数[0], in2 := 8.0)
   END_RUNG wire#w5
   // the same network as SCL:
   #Servo_Instance_2(Axis := "输入轴移载伺服-1",   // "Servo"
                     SON := "急停按钮",
                     Reset := "复位按钮",
                     Mode := 3,
                     MoveHome := "SERVER_DB".工位一移载伺服手动参数[0] = (-1.0),
                     Halt := "程序停止",
                     Position := "SERVER_DB".工位一移载伺服手动参数[2],
                     Velocity := "SERVER_DB".工位一移载伺服手动参数[1],
                     JogForword := "SERVER_DB".工位一移载伺服手动参数[0] = 1.0,
                     JogBackword := "SERVER_DB".工位一移载伺服手动参数[0] = 2.0,
                     MoveAbsolute := "SERVER_DB".工位一移载伺服手动参数[0] = 4.0,
                     MoveRelative := "SERVER_DB".工位一移载伺服手动参数[0] = 8.0);
END_REGION

REGION Network 4: 手动输入轴移载伺服-2
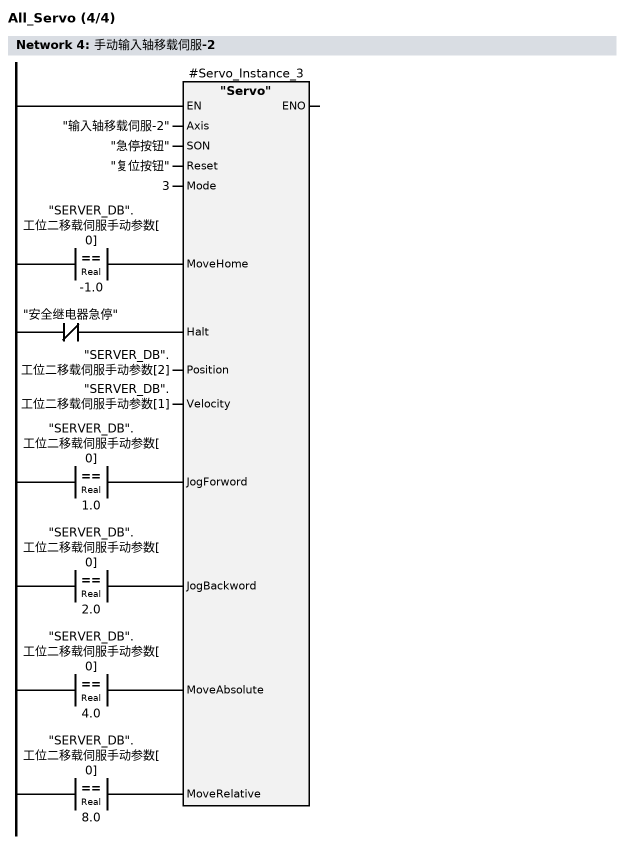
   RUNG wire#powerrail
      #Servo_Instance_3(MoveHome := wire#w1, Halt := wire#w2, JogForword := wire#w3, JogBackword := wire#w4, MoveAbsolute := wire#w5, MoveRelative := wire#w6, Axis := "输入轴移载伺服-2", SON := "急停按钮", Reset := "复位按钮", Mode := 3, Position := "SERVER_DB".工位二移载伺服手动参数[2], Velocity := "SERVER_DB".工位二移载伺服手动参数[1])
   END_RUNG
   RUNG wire#powerrail
      { S7_Templates := "SrcType := Real" } EQ_Contact(in1 := "SERVER_DB".工位二移载伺服手动参数[0], in2 := -1.0)
   END_RUNG wire#w1
   RUNG wire#powerrail
      I_Contact( "安全继电器急停" )
   END_RUNG wire#w2
   RUNG wire#powerrail
      { S7_Templates := "SrcType := Real" } EQ_Contact(in1 := "SERVER_DB".工位二移载伺服手动参数[0], in2 := 1.0)
   END_RUNG wire#w3
   RUNG wire#powerrail
      { S7_Templates := "SrcType := Real" } EQ_Contact(in1 := "SERVER_DB".工位二移载伺服手动参数[0], in2 := 2.0)
   END_RUNG wire#w4
   RUNG wire#powerrail
      { S7_Templates := "SrcType := Real" } EQ_Contact(in1 := "SERVER_DB".工位二移载伺服手动参数[0], in2 := 4.0)
   END_RUNG wire#w5
   RUNG wire#powerrail
      { S7_Templates := "SrcType := Real" } EQ_Contact(in1 := "SERVER_DB".工位二移载伺服手动参数[0], in2 := 8.0)
   END_RUNG wire#w6
   // the same network as SCL:
   #Servo_Instance_3(Axis := "输入轴移载伺服-2",   // "Servo"
                     SON := "急停按钮",
                     Reset := "复位按钮",
                     Mode := 3,
                     MoveHome := "SERVER_DB".工位二移载伺服手动参数[0] = (-1.0),
                     Halt := NOT "安全继电器急停",
                     Position := "SERVER_DB".工位二移载伺服手动参数[2],
                     Velocity := "SERVER_DB".工位二移载伺服手动参数[1],
                     JogForword := "SERVER_DB".工位二移载伺服手动参数[0] = 1.0,
                     JogBackword := "SERVER_DB".工位二移载伺服手动参数[0] = 2.0,
                     MoveAbsolute := "SERVER_DB".工位二移载伺服手动参数[0] = 4.0,
                     MoveRelative := "SERVER_DB".工位二移载伺服手动参数[0] = 8.0);
END_REGION
END_FUNCTION_BLOCK

FUNCTION_BLOCK "Auto2"   // FB3, LAD
{ S7_Optimized_Access := 'TRUE' }
VERSION : 0.1
   VAR
      Temp : Array[0..20] of Bool;
      newCV : DInt;
      MC_Halt_Instance : MC_Halt;
      IEC_Timer_0_Instance : TON_TIME;
      IEC_Timer_0_Instance_1 : TON_TIME;
      MC_MoveAbsolute_Instance : MC_MoveAbsolute;
      MC_MoveAbsolute_Instance_1 : MC_MoveAbsolute;
      MC_MoveAbsolute_Instance_2 : MC_MoveAbsolute;
      MC_MoveRelative_Instance : MC_MoveRelative;
      MC_MoveRelative_Instance_1 : MC_MoveRelative;
      MC_MoveRelative_Instance_2 : MC_MoveRelative;
      MC_MoveRelative_Instance_3 : MC_MoveRelative;
      MC_MoveRelative_Instance_4 : MC_MoveRelative;
      IEC_Timer_0_Instance_2 : TON_TIME;
      IEC_Timer_0_Instance_3 : TON_TIME;
   END_VAR
   VAR RETAIN
      IEC_Counter_0_Instance : CTU_INT;
   END_VAR
   VAR
      CTRL_HSC_0_Instance : CTRL_HSC;
      IEC_Timer_0_Instance_4 : TON_TIME;
      MC_MoveRelative_Instance_5 : MC_MoveRelative;
      工位2输入轴移载夹紧_Instance : "工位2输入轴移载夹紧";
      工位2复检_Instance : "工位2复检";
      工位2复检_Instance_1 : "工位2复检";
      工位2复检_Instance_2 : "工位2复检";
      工位2复检_Instance_3 : "工位2复检";
      工位2复检_Instance_4 : "工位2复检";
      工位2复检_Instance_5 : "工位2复检";
      工位2复位_Instance : "工位2复位";
   END_VAR
   VAR_TEMP   // added for the SCL form of the ladder/FBD networks
      _w1 : Bool;
      _w2 : Bool;
      _w3 : Bool;
   END_VAR
BEGIN

REGION Network 1
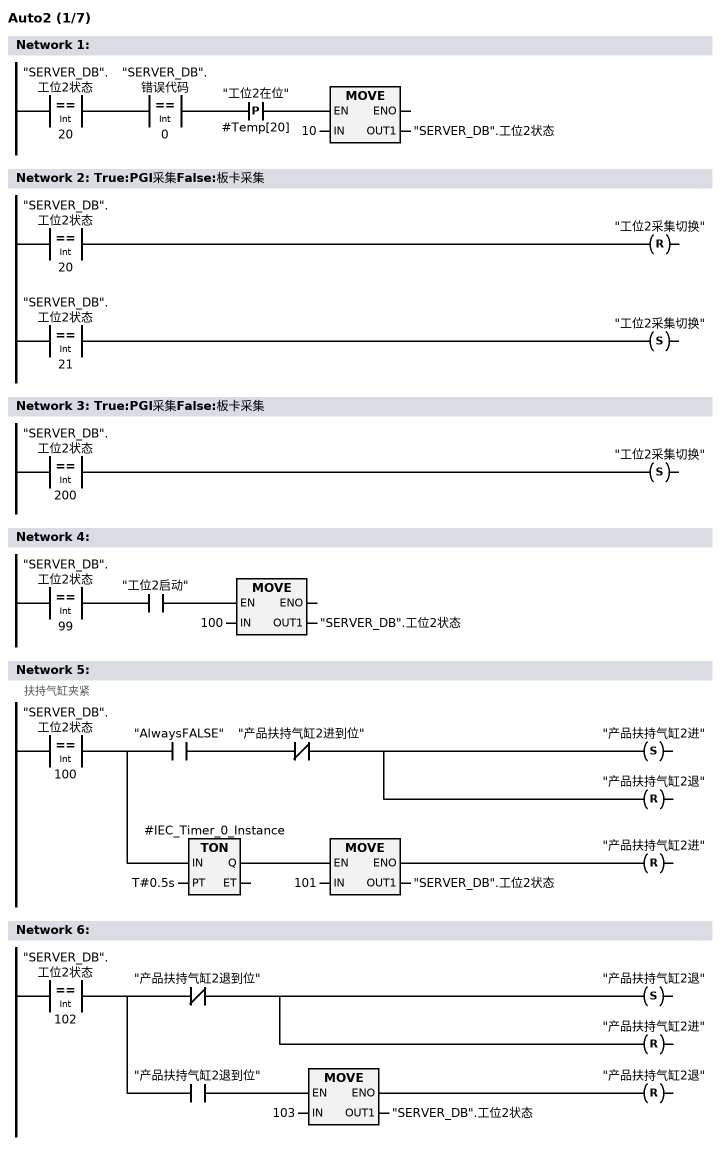
   RUNG wire#powerrail
      { S7_Templates := "SrcType := Int" } EQ_Contact(in1 := "SERVER_DB".工位2状态, in2 := 20)
      { S7_Templates := "SrcType := Int" } EQ_Contact(in1 := "SERVER_DB".错误代码, in2 := 0)
      P_Contact(operand := "工位2在位", bit := #Temp[20])
      Move(in := 10, out1 => "SERVER_DB".工位2状态)
   END_RUNG
   // the same network as SCL:
   #_w1 := ("SERVER_DB".工位2状态 = 20) AND ("SERVER_DB".错误代码 = 0) AND "工位2在位" AND NOT #Temp[20];   // rising edge of "工位2在位"
   #Temp[20] := "工位2在位";
   IF #_w1 THEN "SERVER_DB".工位2状态 := 10; END_IF;
END_REGION

REGION Network 2: True:PGI采集False:板卡采集
   RUNG wire#powerrail
      { S7_Templates := "SrcType := Int" } EQ_Contact(in1 := "SERVER_DB".工位2状态, in2 := 20)
      R_Coil( "工位2采集切换" )
   END_RUNG
   RUNG wire#powerrail
      { S7_Templates := "SrcType := Int" } EQ_Contact(in1 := "SERVER_DB".工位2状态, in2 := 21)
      S_Coil( "工位2采集切换" )
   END_RUNG
   // the same network as SCL:
   IF "SERVER_DB".工位2状态 = 20 THEN "工位2采集切换" := FALSE; END_IF;
   IF "SERVER_DB".工位2状态 = 21 THEN "工位2采集切换" := TRUE; END_IF;
END_REGION

REGION Network 3: True:PGI采集False:板卡采集
   RUNG wire#powerrail
      { S7_Templates := "SrcType := Int" } EQ_Contact(in1 := "SERVER_DB".工位2状态, in2 := 200)
      S_Coil( "工位2采集切换" )
   END_RUNG
   // the same network as SCL:
   IF "SERVER_DB".工位2状态 = 200 THEN "工位2采集切换" := TRUE; END_IF;
END_REGION

REGION Network 4
   RUNG wire#powerrail
      { S7_Templates := "SrcType := Int" } EQ_Contact(in1 := "SERVER_DB".工位2状态, in2 := 99)
      Contact( "工位2启动" )
      Move(in := 100, out1 => "SERVER_DB".工位2状态)
   END_RUNG
   // the same network as SCL:
   IF ("SERVER_DB".工位2状态 = 99) AND "工位2启动" THEN "SERVER_DB".工位2状态 := 100; END_IF;
END_REGION

REGION Network 5
   // 扶持气缸夹紧
   #_w1 := "SERVER_DB".工位2状态 = 100;
   IF #_w1 AND "AlwaysFALSE" AND NOT "产品扶持气缸2进到位" THEN
       "产品扶持气缸2进" := TRUE;
       "产品扶持气缸2退" := FALSE;
   END_IF;
   #IEC_Timer_0_Instance(IN := #_w1, PT := T#0.5s);   // TON
   IF #IEC_Timer_0_Instance.Q THEN
       "SERVER_DB".工位2状态 := 101;
       "产品扶持气缸2进" := FALSE;
   END_IF;
END_REGION

REGION Network 6
   RUNG wire#powerrail
      { S7_Templates := "SrcType := Int" } EQ_Contact(in1 := "SERVER_DB".工位2状态, in2 := 102)
      wire#w1
      I_Contact( "产品扶持气缸2退到位" )
      wire#w2
      S_Coil( "产品扶持气缸2退" )
   END_RUNG
   RUNG wire#w2
      R_Coil( "产品扶持气缸2进" )
   END_RUNG
   RUNG wire#w1
      Contact( "产品扶持气缸2退到位" )
      Move(in := 103, out1 => "SERVER_DB".工位2状态)
      R_Coil( "产品扶持气缸2退" )
   END_RUNG
   // the same network as SCL:
   #_w1 := "SERVER_DB".工位2状态 = 102;
   IF #_w1 AND NOT "产品扶持气缸2退到位" THEN
       "产品扶持气缸2退" := TRUE;
       "产品扶持气缸2进" := FALSE;
   END_IF;
   IF #_w1 AND "产品扶持气缸2退到位" THEN
       "SERVER_DB".工位2状态 := 103;
       "产品扶持气缸2退" := FALSE;
   END_IF;
END_REGION

REGION Network 7
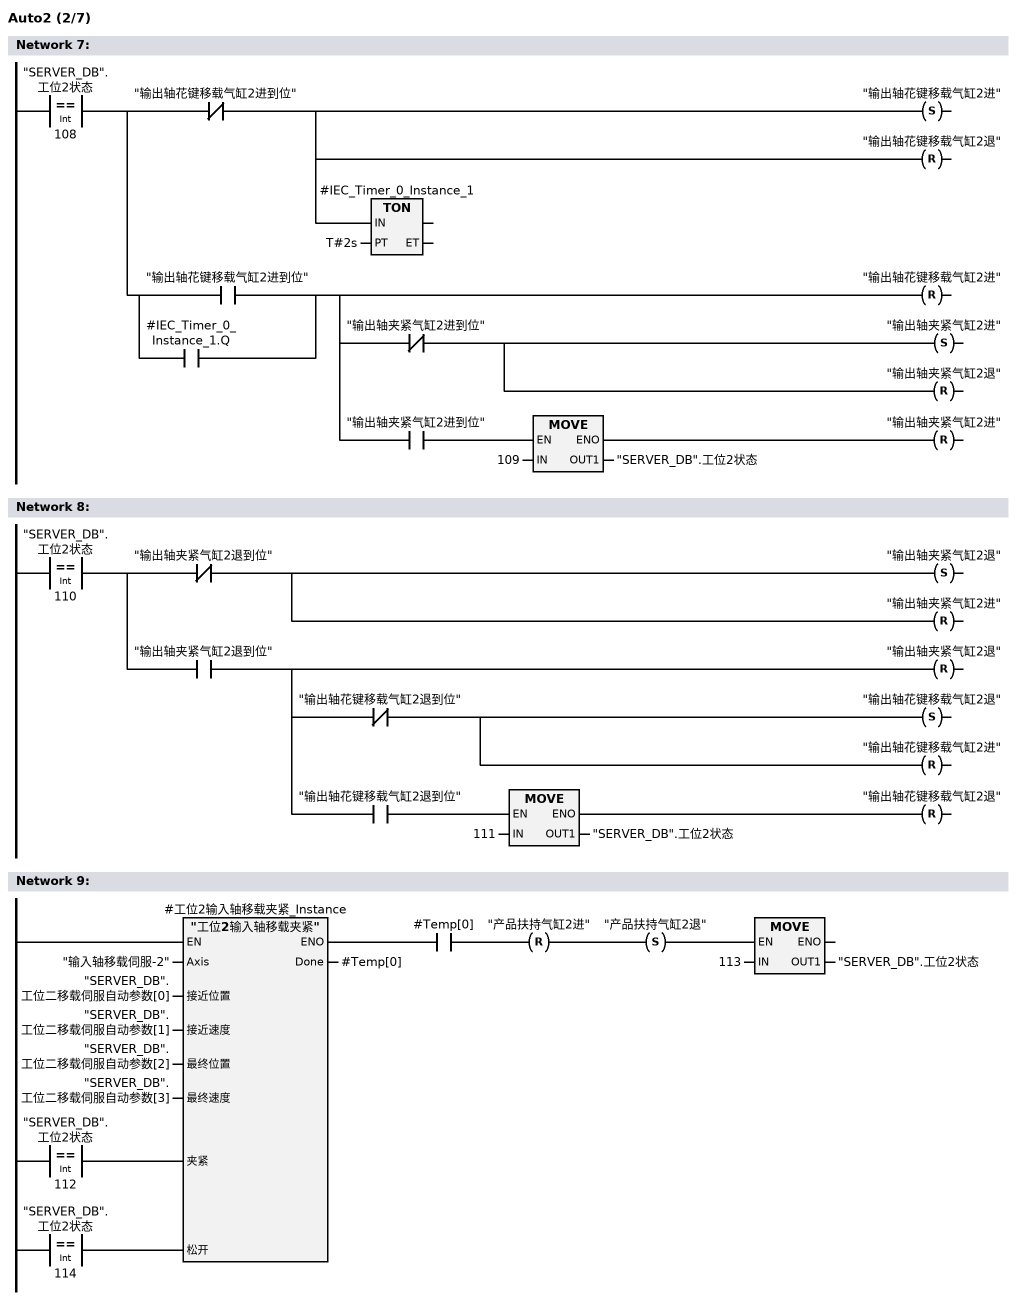
   #_w1 := "SERVER_DB".工位2状态 = 108;
   #_w2 := #_w1 AND NOT "输出轴花键移载气缸2进到位";
   IF #_w2 THEN
       "输出轴花键移载气缸2进" := TRUE;
       "输出轴花键移载气缸2退" := FALSE;
   END_IF;
   #IEC_Timer_0_Instance_1(IN := #_w2, PT := T#2s);   // TON
   #_w3 := #_w1 AND ("输出轴花键移载气缸2进到位" OR #IEC_Timer_0_Instance_1.Q);
   IF #_w3 THEN "输出轴花键移载气缸2进" := FALSE; END_IF;
   IF #_w3 AND NOT "输出轴夹紧气缸2进到位" THEN
       "输出轴夹紧气缸2进" := TRUE;
       "输出轴夹紧气缸2退" := FALSE;
   END_IF;
   IF #_w3 AND "输出轴夹紧气缸2进到位" THEN
       "SERVER_DB".工位2状态 := 109;
       "输出轴夹紧气缸2进" := FALSE;
   END_IF;
END_REGION

REGION Network 8
   RUNG wire#powerrail
      { S7_Templates := "SrcType := Int" } EQ_Contact(in1 := "SERVER_DB".工位2状态, in2 := 110)
      wire#w1
      I_Contact( "输出轴夹紧气缸2退到位" )
      wire#w2
      S_Coil( "输出轴夹紧气缸2退" )
   END_RUNG
   RUNG wire#w2
      R_Coil( "输出轴夹紧气缸2进" )
   END_RUNG
   RUNG wire#w1
      Contact( "输出轴夹紧气缸2退到位" )
      wire#w3
      R_Coil( "输出轴夹紧气缸2退" )
   END_RUNG
   RUNG wire#w3
      I_Contact( "输出轴花键移载气缸2退到位" )
      wire#w4
      S_Coil( "输出轴花键移载气缸2退" )
   END_RUNG
   RUNG wire#w4
      R_Coil( "输出轴花键移载气缸2进" )
   END_RUNG
   RUNG wire#w3
      Contact( "输出轴花键移载气缸2退到位" )
      Move(in := 111, out1 => "SERVER_DB".工位2状态)
      R_Coil( "输出轴花键移载气缸2退" )
   END_RUNG
   // the same network as SCL:
   #_w1 := "SERVER_DB".工位2状态 = 110;
   IF #_w1 AND NOT "输出轴夹紧气缸2退到位" THEN
       "输出轴夹紧气缸2退" := TRUE;
       "输出轴夹紧气缸2进" := FALSE;
   END_IF;
   #_w2 := #_w1 AND "输出轴夹紧气缸2退到位";
   IF #_w2 THEN "输出轴夹紧气缸2退" := FALSE; END_IF;
   IF #_w2 AND NOT "输出轴花键移载气缸2退到位" THEN
       "输出轴花键移载气缸2退" := TRUE;
       "输出轴花键移载气缸2进" := FALSE;
   END_IF;
   IF #_w2 AND "输出轴花键移载气缸2退到位" THEN
       "SERVER_DB".工位2状态 := 111;
       "输出轴花键移载气缸2退" := FALSE;
   END_IF;
END_REGION

REGION Network 9
   RUNG wire#powerrail
      #工位2输入轴移载夹紧_Instance(夹紧 := wire#w1, 松开 := wire#w2, Axis := "输入轴移载伺服-2", 接近位置 := "SERVER_DB".工位二移载伺服自动参数[0], 接近速度 := "SERVER_DB".工位二移载伺服自动参数[1], 最终位置 := "SERVER_DB".工位二移载伺服自动参数[2], 最终速度 := "SERVER_DB".工位二移载伺服自动参数[3], Done => #Temp[0])
      Contact( #Temp[0] )
      R_Coil( "产品扶持气缸2进" )
      S_Coil( "产品扶持气缸2退" )
      Move(in := 113, out1 => "SERVER_DB".工位2状态)
   END_RUNG
   RUNG wire#powerrail
      { S7_Templates := "SrcType := Int" } EQ_Contact(in1 := "SERVER_DB".工位2状态, in2 := 112)
   END_RUNG wire#w1
   RUNG wire#powerrail
      { S7_Templates := "SrcType := Int" } EQ_Contact(in1 := "SERVER_DB".工位2状态, in2 := 114)
   END_RUNG wire#w2
   // the same network as SCL:
   #工位2输入轴移载夹紧_Instance(Axis := "输入轴移载伺服-2",   // "工位2输入轴移载夹紧"
                        接近位置 := "SERVER_DB".工位二移载伺服自动参数[0],
                        接近速度 := "SERVER_DB".工位二移载伺服自动参数[1],
                        最终位置 := "SERVER_DB".工位二移载伺服自动参数[2],
                        最终速度 := "SERVER_DB".工位二移载伺服自动参数[3],
                        夹紧 := "SERVER_DB".工位2状态 = 112,
                        松开 := "SERVER_DB".工位2状态 = 114,
                        Done => #Temp[0],
                        ENO => #_w1);
   IF #_w1 AND #Temp[0] THEN
       "产品扶持气缸2进" := FALSE;
       "产品扶持气缸2退" := TRUE;
       "SERVER_DB".工位2状态 := 113;
   END_IF;
END_REGION

REGION Network 10: True:板卡供电False:PGI供电
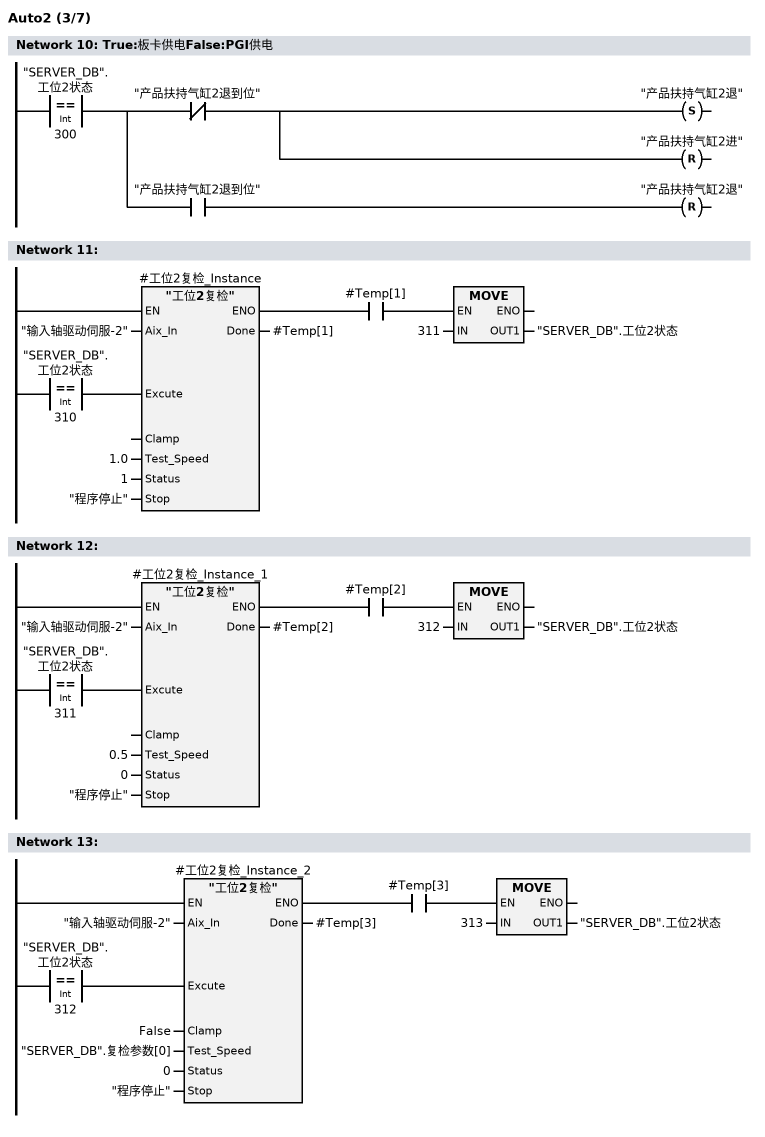
   RUNG wire#powerrail
      { S7_Templates := "SrcType := Int" } EQ_Contact(in1 := "SERVER_DB".工位2状态, in2 := 300)
      wire#w1
      I_Contact( "产品扶持气缸2退到位" )
      wire#w2
      S_Coil( "产品扶持气缸2退" )
   END_RUNG
   RUNG wire#w2
      R_Coil( "产品扶持气缸2进" )
   END_RUNG
   RUNG wire#w1
      Contact( "产品扶持气缸2退到位" )
      R_Coil( "产品扶持气缸2退" )
   END_RUNG
   // the same network as SCL:
   #_w1 := "SERVER_DB".工位2状态 = 300;
   IF #_w1 AND NOT "产品扶持气缸2退到位" THEN
       "产品扶持气缸2退" := TRUE;
       "产品扶持气缸2进" := FALSE;
   END_IF;
   IF #_w1 AND "产品扶持气缸2退到位" THEN "产品扶持气缸2退" := FALSE; END_IF;
END_REGION

REGION Network 11
   RUNG wire#powerrail
      #工位2复检_Instance(Excute := wire#w1, Aix_In := "输入轴驱动伺服-2", Clamp :=, Test_Speed := 1.0, Status := 1, Stop := "程序停止", Done => #Temp[1])
      Contact( #Temp[1] )
      Move(in := 311, out1 => "SERVER_DB".工位2状态)
   END_RUNG
   RUNG wire#powerrail
      { S7_Templates := "SrcType := Int" } EQ_Contact(in1 := "SERVER_DB".工位2状态, in2 := 310)
   END_RUNG wire#w1
   // the same network as SCL:
   #工位2复检_Instance(Aix_In := "输入轴驱动伺服-2",   // "工位2复检"
                   Excute := "SERVER_DB".工位2状态 = 310,
                   Test_Speed := 1.0,
                   Status := 1,
                   Stop := "程序停止",
                   Done => #Temp[1],
                   ENO => #_w1);
   IF #_w1 AND #Temp[1] THEN "SERVER_DB".工位2状态 := 311; END_IF;
END_REGION

REGION Network 12
   RUNG wire#powerrail
      #工位2复检_Instance_1(Excute := wire#w1, Aix_In := "输入轴驱动伺服-2", Clamp :=, Test_Speed := 0.5, Status := 0, Stop := "程序停止", Done => #Temp[2])
      Contact( #Temp[2] )
      Move(in := 312, out1 => "SERVER_DB".工位2状态)
   END_RUNG
   RUNG wire#powerrail
      { S7_Templates := "SrcType := Int" } EQ_Contact(in1 := "SERVER_DB".工位2状态, in2 := 311)
   END_RUNG wire#w1
   // the same network as SCL:
   #工位2复检_Instance_1(Aix_In := "输入轴驱动伺服-2",   // "工位2复检"
                     Excute := "SERVER_DB".工位2状态 = 311,
                     Test_Speed := 0.5,
                     Status := 0,
                     Stop := "程序停止",
                     Done => #Temp[2],
                     ENO => #_w1);
   IF #_w1 AND #Temp[2] THEN "SERVER_DB".工位2状态 := 312; END_IF;
END_REGION

REGION Network 13
   RUNG wire#powerrail
      #工位2复检_Instance_2(Excute := wire#w1, Aix_In := "输入轴驱动伺服-2", Clamp := False, Test_Speed := "SERVER_DB".复检参数[0], Status := 0, Stop := "程序停止", Done => #Temp[3])
      Contact( #Temp[3] )
      Move(in := 313, out1 => "SERVER_DB".工位2状态)
   END_RUNG
   RUNG wire#powerrail
      { S7_Templates := "SrcType := Int" } EQ_Contact(in1 := "SERVER_DB".工位2状态, in2 := 312)
   END_RUNG wire#w1
   // the same network as SCL:
   #工位2复检_Instance_2(Aix_In := "输入轴驱动伺服-2",   // "工位2复检"
                     Excute := "SERVER_DB".工位2状态 = 312,
                     Clamp := False,
                     Test_Speed := "SERVER_DB".复检参数[0],
                     Status := 0,
                     Stop := "程序停止",
                     Done => #Temp[3],
                     ENO => #_w1);
   IF #_w1 AND #Temp[3] THEN "SERVER_DB".工位2状态 := 313; END_IF;
END_REGION

REGION Network 14
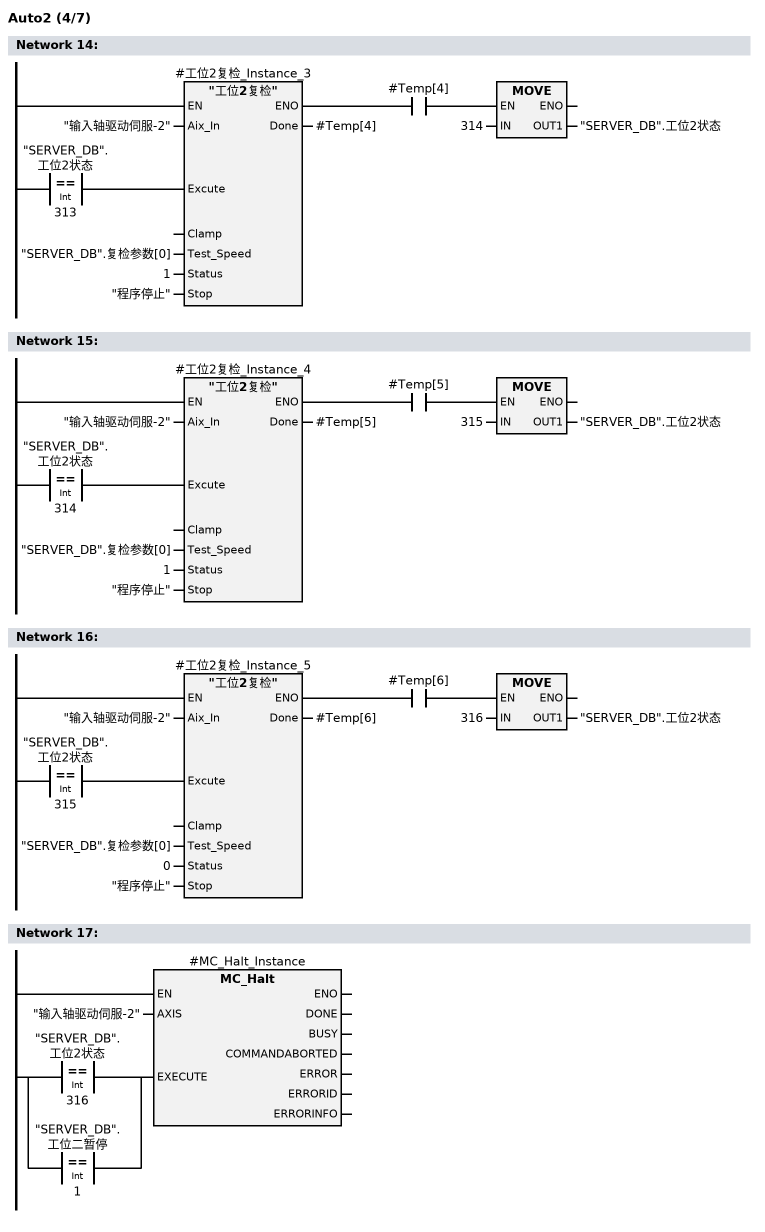
   RUNG wire#powerrail
      #工位2复检_Instance_3(Excute := wire#w1, Aix_In := "输入轴驱动伺服-2", Clamp :=, Test_Speed := "SERVER_DB".复检参数[0], Status := 1, Stop := "程序停止", Done => #Temp[4])
      Contact( #Temp[4] )
      Move(in := 314, out1 => "SERVER_DB".工位2状态)
   END_RUNG
   RUNG wire#powerrail
      { S7_Templates := "SrcType := Int" } EQ_Contact(in1 := "SERVER_DB".工位2状态, in2 := 313)
   END_RUNG wire#w1
   // the same network as SCL:
   #工位2复检_Instance_3(Aix_In := "输入轴驱动伺服-2",   // "工位2复检"
                     Excute := "SERVER_DB".工位2状态 = 313,
                     Test_Speed := "SERVER_DB".复检参数[0],
                     Status := 1,
                     Stop := "程序停止",
                     Done => #Temp[4],
                     ENO => #_w1);
   IF #_w1 AND #Temp[4] THEN "SERVER_DB".工位2状态 := 314; END_IF;
END_REGION

REGION Network 15
   RUNG wire#powerrail
      #工位2复检_Instance_4(Excute := wire#w1, Aix_In := "输入轴驱动伺服-2", Clamp :=, Test_Speed := "SERVER_DB".复检参数[0], Status := 1, Stop := "程序停止", Done => #Temp[5])
      Contact( #Temp[5] )
      Move(in := 315, out1 => "SERVER_DB".工位2状态)
   END_RUNG
   RUNG wire#powerrail
      { S7_Templates := "SrcType := Int" } EQ_Contact(in1 := "SERVER_DB".工位2状态, in2 := 314)
   END_RUNG wire#w1
   // the same network as SCL:
   #工位2复检_Instance_4(Aix_In := "输入轴驱动伺服-2",   // "工位2复检"
                     Excute := "SERVER_DB".工位2状态 = 314,
                     Test_Speed := "SERVER_DB".复检参数[0],
                     Status := 1,
                     Stop := "程序停止",
                     Done => #Temp[5],
                     ENO => #_w1);
   IF #_w1 AND #Temp[5] THEN "SERVER_DB".工位2状态 := 315; END_IF;
END_REGION

REGION Network 16
   RUNG wire#powerrail
      #工位2复检_Instance_5(Excute := wire#w1, Aix_In := "输入轴驱动伺服-2", Clamp :=, Test_Speed := "SERVER_DB".复检参数[0], Status := 0, Stop := "程序停止", Done => #Temp[6])
      Contact( #Temp[6] )
      Move(in := 316, out1 => "SERVER_DB".工位2状态)
   END_RUNG
   RUNG wire#powerrail
      { S7_Templates := "SrcType := Int" } EQ_Contact(in1 := "SERVER_DB".工位2状态, in2 := 315)
   END_RUNG wire#w1
   // the same network as SCL:
   #工位2复检_Instance_5(Aix_In := "输入轴驱动伺服-2",   // "工位2复检"
                     Excute := "SERVER_DB".工位2状态 = 315,
                     Test_Speed := "SERVER_DB".复检参数[0],
                     Status := 0,
                     Stop := "程序停止",
                     Done => #Temp[6],
                     ENO => #_w1);
   IF #_w1 AND #Temp[6] THEN "SERVER_DB".工位2状态 := 316; END_IF;
END_REGION

REGION Network 17
   #MC_Halt_Instance(Axis := "输入轴驱动伺服-2", Execute := ("SERVER_DB".工位2状态 = 316) OR ("SERVER_DB".工位二暂停 = 1));   // MC_Halt
END_REGION

REGION Network 18
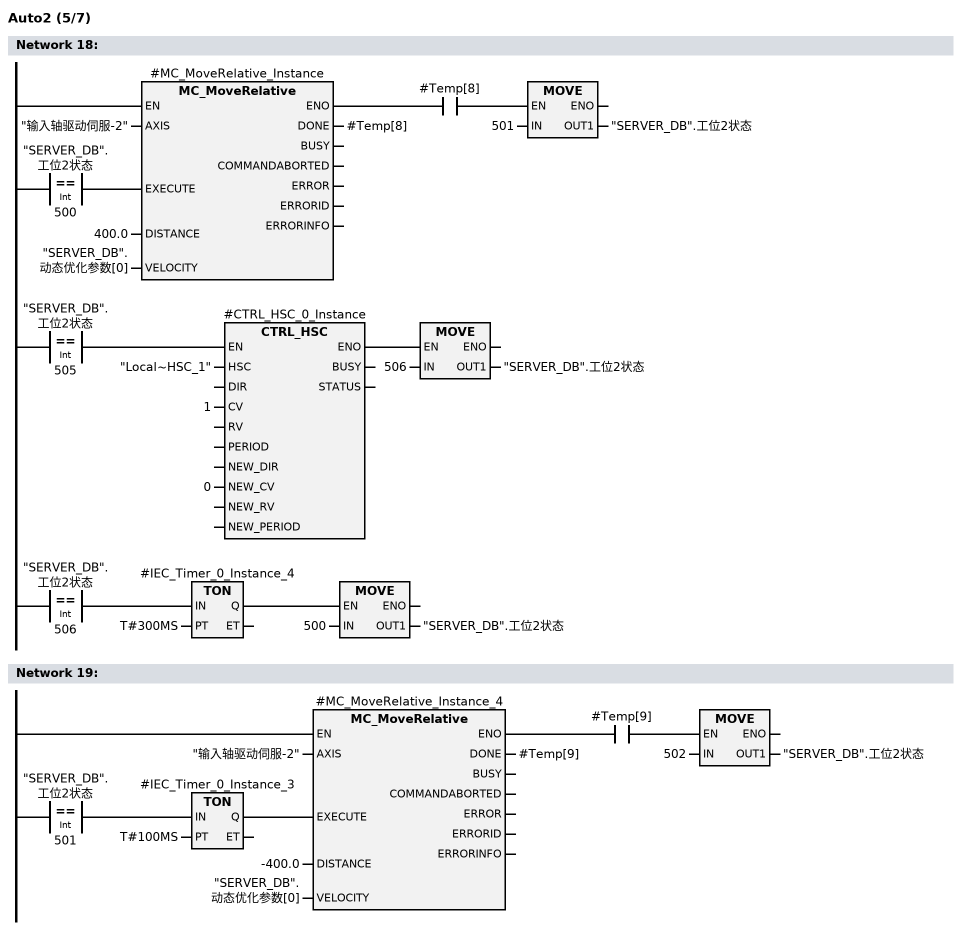
   // ENO of a box is taken as its EN; it also drops when the box reports an error
   #MC_MoveRelative_Instance(Axis := "输入轴驱动伺服-2",   // MC_MoveRelative
                           Execute := "SERVER_DB".工位2状态 = 500,
                           Distance := 400.0,
                           Velocity := "SERVER_DB".动态优化参数[0],
                           Done => #Temp[8]);
   IF #Temp[8] THEN "SERVER_DB".工位2状态 := 501; END_IF;
   #_w1 := "SERVER_DB".工位2状态 = 505;
   IF #_w1 THEN
       #CTRL_HSC_0_Instance(HSC := "Local~HSC_1", CV := 1, NEW_CV := 0);   // CTRL_HSC
       "SERVER_DB".工位2状态 := 506;
   END_IF;
   #IEC_Timer_0_Instance_4(IN := "SERVER_DB".工位2状态 = 506, PT := T#300MS);   // TON
   IF #IEC_Timer_0_Instance_4.Q THEN "SERVER_DB".工位2状态 := 500; END_IF;
END_REGION

REGION Network 19
   // ENO of a box is taken as its EN; it also drops when the box reports an error
   #IEC_Timer_0_Instance_3(IN := "SERVER_DB".工位2状态 = 501, PT := T#100MS);   // TON
   #MC_MoveRelative_Instance_4(Axis := "输入轴驱动伺服-2",   // MC_MoveRelative
                           Execute := #IEC_Timer_0_Instance_3.Q,
                           Distance := -400.0,
                           Velocity := "SERVER_DB".动态优化参数[0],
                           Done => #Temp[9]);
   IF #Temp[9] THEN "SERVER_DB".工位2状态 := 502; END_IF;
END_REGION

REGION Network 20
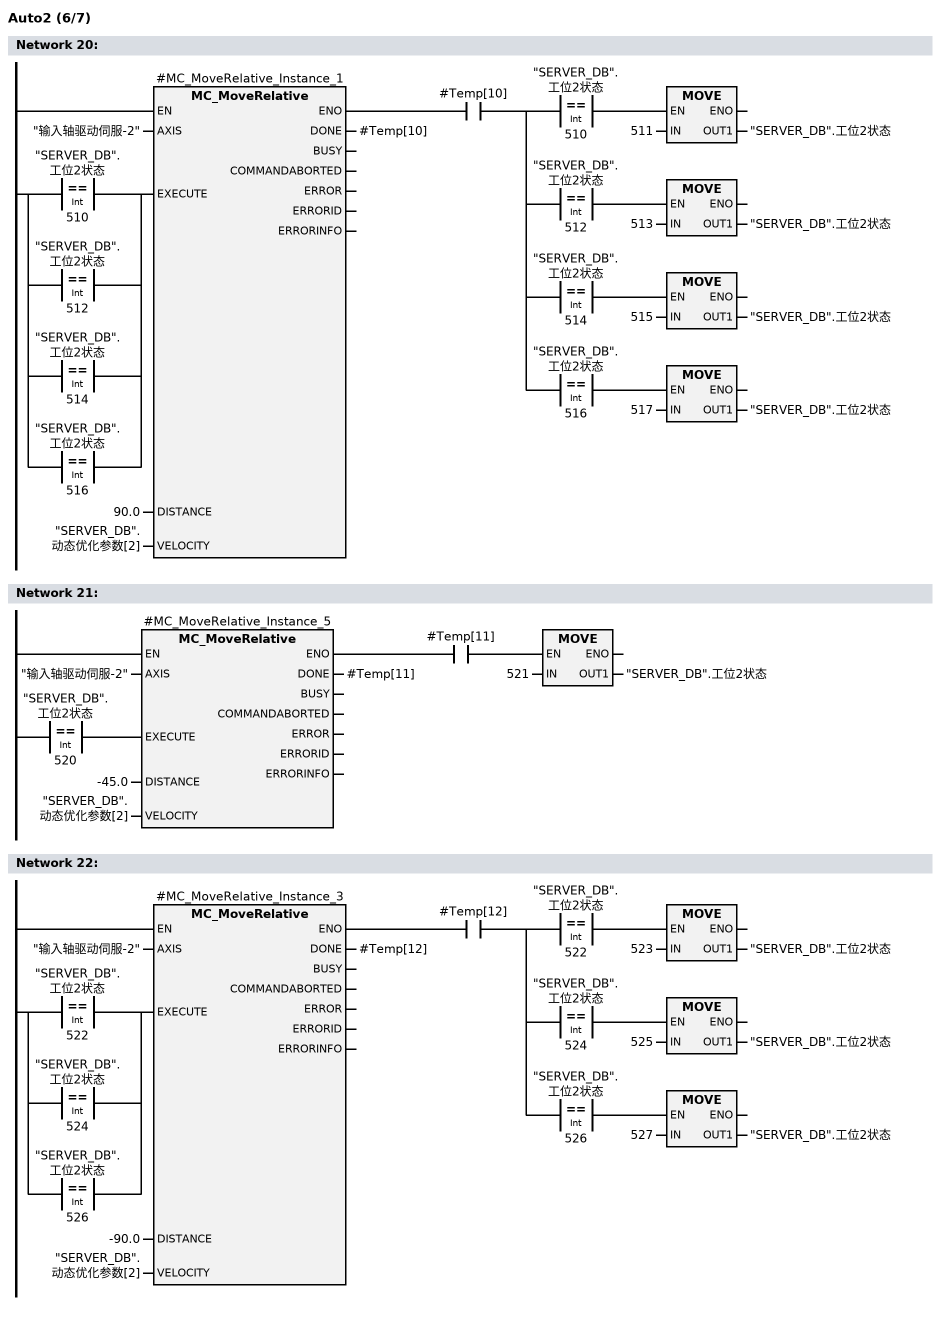
   // ENO of a box is taken as its EN; it also drops when the box reports an error
   #MC_MoveRelative_Instance_1(Axis := "输入轴驱动伺服-2",   // MC_MoveRelative
                           Execute := ("SERVER_DB".工位2状态 = 510) OR ("SERVER_DB".工位2状态 = 512) OR ("SERVER_DB".工位2状态 = 514) OR ("SERVER_DB".工位2状态 = 516),
                           Distance := 90.0,
                           Velocity := "SERVER_DB".动态优化参数[2],
                           Done => #Temp[10]);
   IF #Temp[10] AND ("SERVER_DB".工位2状态 = 510) THEN "SERVER_DB".工位2状态 := 511; END_IF;
   IF #Temp[10] AND ("SERVER_DB".工位2状态 = 512) THEN "SERVER_DB".工位2状态 := 513; END_IF;
   IF #Temp[10] AND ("SERVER_DB".工位2状态 = 514) THEN "SERVER_DB".工位2状态 := 515; END_IF;
   IF #Temp[10] AND ("SERVER_DB".工位2状态 = 516) THEN "SERVER_DB".工位2状态 := 517; END_IF;
END_REGION

REGION Network 21
   // ENO of a box is taken as its EN; it also drops when the box reports an error
   #MC_MoveRelative_Instance_5(Axis := "输入轴驱动伺服-2",   // MC_MoveRelative
                           Execute := "SERVER_DB".工位2状态 = 520,
                           Distance := -45.0,
                           Velocity := "SERVER_DB".动态优化参数[2],
                           Done => #Temp[11]);
   IF #Temp[11] THEN "SERVER_DB".工位2状态 := 521; END_IF;
END_REGION

REGION Network 22
   // ENO of a box is taken as its EN; it also drops when the box reports an error
   #MC_MoveRelative_Instance_3(Axis := "输入轴驱动伺服-2",   // MC_MoveRelative
                           Execute := ("SERVER_DB".工位2状态 = 522) OR ("SERVER_DB".工位2状态 = 524) OR ("SERVER_DB".工位2状态 = 526),
                           Distance := -90.0,
                           Velocity := "SERVER_DB".动态优化参数[2],
                           Done => #Temp[12]);
   IF #Temp[12] AND ("SERVER_DB".工位2状态 = 522) THEN "SERVER_DB".工位2状态 := 523; END_IF;
   IF #Temp[12] AND ("SERVER_DB".工位2状态 = 524) THEN "SERVER_DB".工位2状态 := 525; END_IF;
   IF #Temp[12] AND ("SERVER_DB".工位2状态 = 526) THEN "SERVER_DB".工位2状态 := 527; END_IF;
END_REGION

REGION Network 23
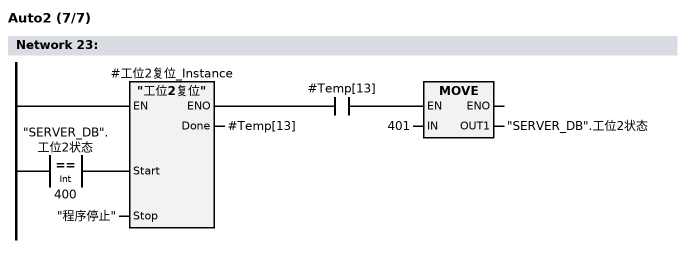
   RUNG wire#powerrail
      #工位2复位_Instance(Start := wire#w1, Stop := "程序停止", Done => #Temp[13])
      Contact( #Temp[13] )
      Move(in := 401, out1 => "SERVER_DB".工位2状态)
   END_RUNG
   RUNG wire#powerrail
      { S7_Templates := "SrcType := Int" } EQ_Contact(in1 := "SERVER_DB".工位2状态, in2 := 400)
   END_RUNG wire#w1
   // the same network as SCL:
   #工位2复位_Instance(Start := "SERVER_DB".工位2状态 = 400, Stop := "程序停止", Done => #Temp[13], ENO => #_w1);   // "工位2复位"
   IF #_w1 AND #Temp[13] THEN "SERVER_DB".工位2状态 := 401; END_IF;
END_REGION
END_FUNCTION_BLOCK

FUNCTION_BLOCK "工位1复检"   // FB4, LAD
{ S7_Optimized_Access := 'TRUE' }
VERSION : 0.1
   VAR_INPUT
      Aix_In : TO_PositioningAxis;
      Excute : Bool;
      Clamp : Bool;
      Test_Speed : Real;
      Status : Byte;
      Stop : Bool;
   END_VAR
   VAR_OUTPUT
      Done : Bool;
   END_VAR
   VAR
      "Step" : Int;
      Test_Velocity : Real;
      Temp : Array[0..7] of Bool;
      MC_Halt_Instance : MC_Halt;
      MC_MoveVelocity_Instance : MC_MoveVelocity;
      MC_Halt_Instance_1 : MC_Halt;
      IEC_Timer_0_Instance : TON_TIME;
      输入轴二次夹紧_Instance : "工位1输入轴二次夹紧";
   END_VAR
   VAR_TEMP   // added for the SCL form of the ladder/FBD networks
      _w1 : Bool;
      _w2 : Bool;
   END_VAR
BEGIN

REGION Network 1
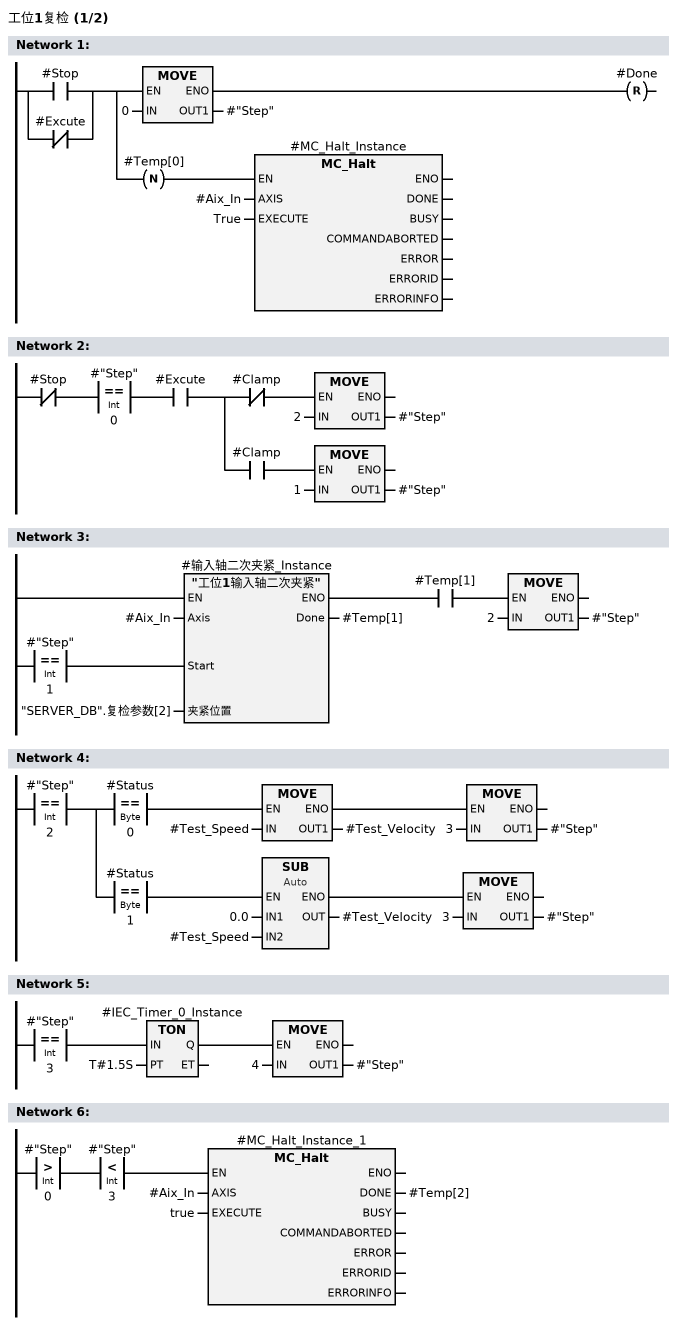
   #_w1 := #Stop OR NOT #Excute;
   IF #_w1 THEN
       #"Step" := 0;
       #Done := FALSE;
   END_IF;
   #_w2 := NOT #_w1 AND #Temp[0];   // falling edge
   #Temp[0] := #_w1;
   IF #_w2 THEN
       #MC_Halt_Instance(Axis := #Aix_In, Execute := True);   // MC_Halt
   END_IF;
END_REGION

REGION Network 2
   RUNG wire#powerrail
      I_Contact( #Stop )
      { S7_Templates := "SrcType := Int" } EQ_Contact(in1 := #"Step", in2 := 0)
      Contact( #Excute )
      wire#w1
      I_Contact( #Clamp )
      Move(in := 2, out1 => #"Step")
   END_RUNG
   RUNG wire#w1
      Contact( #Clamp )
      Move(in := 1, out1 => #"Step")
   END_RUNG
   // the same network as SCL:
   #_w1 := NOT #Stop AND (#"Step" = 0) AND #Excute;
   IF #_w1 AND NOT #Clamp THEN #"Step" := 2; END_IF;
   IF #_w1 AND #Clamp THEN #"Step" := 1; END_IF;
END_REGION

REGION Network 3
   RUNG wire#powerrail
      #输入轴二次夹紧_Instance(Start := wire#w1, Axis := #Aix_In, 夹紧位置 := "SERVER_DB".复检参数[2], Done => #Temp[1])
      Contact( #Temp[1] )
      Move(in := 2, out1 => #"Step")
   END_RUNG
   RUNG wire#powerrail
      { S7_Templates := "SrcType := Int" } EQ_Contact(in1 := #"Step", in2 := 1)
   END_RUNG wire#w1
   // the same network as SCL:
   #输入轴二次夹紧_Instance(Axis := #Aix_In,   // "工位1输入轴二次夹紧"
                     Start := #"Step" = 1,
                     夹紧位置 := "SERVER_DB".复检参数[2],
                     Done => #Temp[1],
                     ENO => #_w1);
   IF #_w1 AND #Temp[1] THEN #"Step" := 2; END_IF;
END_REGION

REGION Network 4
   RUNG wire#powerrail
      { S7_Templates := "SrcType := Int" } EQ_Contact(in1 := #"Step", in2 := 2)
      wire#w1
      { S7_Templates := "SrcType := Byte" } EQ_Contact(in1 := #Status, in2 := 0)
      Move(in := #Test_Speed, out1 => #Test_Velocity)
      Move(in := 3, out1 => #"Step")
   END_RUNG
   RUNG wire#w1
      { S7_Templates := "SrcType := Byte" } EQ_Contact(in1 := #Status, in2 := 1)
      Sub(in1 := 0.0, in2 := #Test_Speed, out => #Test_Velocity)
      Move(in := 3, out1 => #"Step")
   END_RUNG
   // the same network as SCL:
   #_w1 := #"Step" = 2;
   IF #_w1 AND (#Status = 0) THEN
       #Test_Velocity := #Test_Speed;
       #"Step" := 3;
   END_IF;
   IF #_w1 AND (#Status = 1) THEN
       #Test_Velocity := 0.0 - #Test_Speed;
       #"Step" := 3;
   END_IF;
END_REGION

REGION Network 5
   #IEC_Timer_0_Instance(IN := #"Step" = 3, PT := T#1.5S);   // TON
   IF #IEC_Timer_0_Instance.Q THEN #"Step" := 4; END_IF;
END_REGION

REGION Network 6
   IF (#"Step" > 0) AND (#"Step" < 3) THEN
       #MC_Halt_Instance_1(Axis := #Aix_In, Execute := true, Done => #Temp[2]);   // MC_Halt
   END_IF;
END_REGION

REGION Network 7
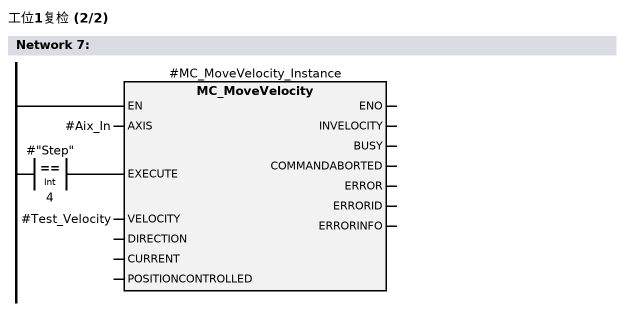
   #MC_MoveVelocity_Instance(Axis := #Aix_In, Execute := #"Step" = 4, Velocity := #Test_Velocity);   // MC_MoveVelocity
END_REGION
END_FUNCTION_BLOCK

FUNCTION_BLOCK "Reset"   // FB5, LAD
{ S7_Optimized_Access := 'TRUE' }
VERSION : 0.1
   VAR_INPUT
      Start : Bool;
      Stop : Bool;
   END_VAR
   VAR_OUTPUT
      Done : Bool;
   END_VAR
   VAR
      "Step" : Int;
      Temp : Array[0..10] of Bool;
      MC_Home_Instance : MC_Home;
      MC_Home_Instance_1 : MC_Home;
      工位2复位_Instance : "工位2复位";
      工位1复位_Instance : "工位1复位";
   END_VAR
   VAR_TEMP   // added for the SCL form of the ladder/FBD networks
      _w1 : Bool;
   END_VAR
BEGIN

REGION Network 1
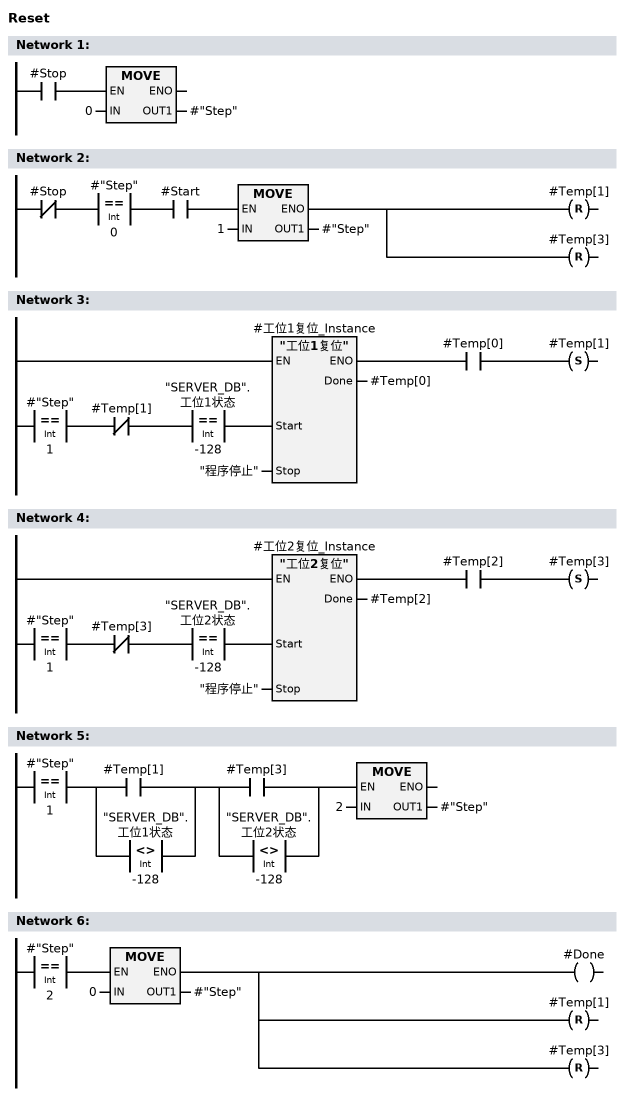
   RUNG wire#powerrail
      Contact( #Stop )
      Move(in := 0, out1 => #"Step")
   END_RUNG
   // the same network as SCL:
   IF #Stop THEN #"Step" := 0; END_IF;
END_REGION

REGION Network 2
   RUNG wire#powerrail
      I_Contact( #Stop )
      { S7_Templates := "SrcType := Int" } EQ_Contact(in1 := #"Step", in2 := 0)
      Contact( #Start )
      Move(in := 1, out1 => #"Step")
      wire#w1
      R_Coil( #Temp[1] )
   END_RUNG
   RUNG wire#w1
      R_Coil( #Temp[3] )
   END_RUNG
   // the same network as SCL:
   #_w1 := NOT #Stop AND (#"Step" = 0) AND #Start;
   IF #_w1 THEN
       #"Step" := 1;
       #Temp[1] := FALSE;
       #Temp[3] := FALSE;
   END_IF;
END_REGION

REGION Network 3
   RUNG wire#powerrail
      #工位1复位_Instance(Start := wire#w1, Stop := "程序停止", Done => #Temp[0])
      Contact( #Temp[0] )
      S_Coil( #Temp[1] )
   END_RUNG
   RUNG wire#powerrail
      { S7_Templates := "SrcType := Int" } EQ_Contact(in1 := #"Step", in2 := 1)
      I_Contact( #Temp[1] )
      { S7_Templates := "SrcType := Int" } EQ_Contact(in1 := "SERVER_DB".工位1状态, in2 := -128)
   END_RUNG wire#w1
   // the same network as SCL:
   #工位1复位_Instance(Start := (#"Step" = 1) AND NOT #Temp[1] AND ("SERVER_DB".工位1状态 = (-128)),   // "工位1复位"
                   Stop := "程序停止",
                   Done => #Temp[0],
                   ENO => #_w1);
   IF #_w1 AND #Temp[0] THEN #Temp[1] := TRUE; END_IF;
END_REGION

REGION Network 4
   RUNG wire#powerrail
      #工位2复位_Instance(Start := wire#w1, Stop := "程序停止", Done => #Temp[2])
      Contact( #Temp[2] )
      S_Coil( #Temp[3] )
   END_RUNG
   RUNG wire#powerrail
      { S7_Templates := "SrcType := Int" } EQ_Contact(in1 := #"Step", in2 := 1)
      I_Contact( #Temp[3] )
      { S7_Templates := "SrcType := Int" } EQ_Contact(in1 := "SERVER_DB".工位2状态, in2 := -128)
   END_RUNG wire#w1
   // the same network as SCL:
   #工位2复位_Instance(Start := (#"Step" = 1) AND NOT #Temp[3] AND ("SERVER_DB".工位2状态 = (-128)),   // "工位2复位"
                   Stop := "程序停止",
                   Done => #Temp[2],
                   ENO => #_w1);
   IF #_w1 AND #Temp[2] THEN #Temp[3] := TRUE; END_IF;
END_REGION

REGION Network 5
   RUNG wire#powerrail
      { S7_Templates := "SrcType := Int" } EQ_Contact(in1 := #"Step", in2 := 1)
      wire#w1
      Contact( #Temp[1] )
      wire#w2
      Contact( #Temp[3] )
      wire#w3
      Move(in := 2, out1 => #"Step")
   END_RUNG
   RUNG wire#w1
      { S7_Templates := "SrcType := Int" } NE_Contact(in1 := "SERVER_DB".工位1状态, in2 := -128)
   END_RUNG wire#w2
   RUNG wire#w2
      { S7_Templates := "SrcType := Int" } NE_Contact(in1 := "SERVER_DB".工位2状态, in2 := -128)
   END_RUNG wire#w3
   // the same network as SCL:
   IF (#"Step" = 1) AND (#Temp[1] OR ("SERVER_DB".工位1状态 <> (-128))) AND (#Temp[3] OR ("SERVER_DB".工位2状态 <> (-128))) THEN
       #"Step" := 2;
   END_IF;
END_REGION

REGION Network 6
   RUNG wire#powerrail
      { S7_Templates := "SrcType := Int" } EQ_Contact(in1 := #"Step", in2 := 2)
      Move(in := 0, out1 => #"Step")
      wire#w1
      Coil( #Done )
   END_RUNG
   RUNG wire#w1
      R_Coil( #Temp[1] )
   END_RUNG
   RUNG wire#w1
      R_Coil( #Temp[3] )
   END_RUNG
   // the same network as SCL:
   #_w1 := #"Step" = 2;
   IF #_w1 THEN #"Step" := 0; END_IF;
   #Done := #_w1;
   IF #_w1 THEN
       #Temp[1] := FALSE;
       #Temp[3] := FALSE;
   END_IF;
END_REGION
END_FUNCTION_BLOCK

FUNCTION_BLOCK "工位1复位"   // FB6, LAD
{ S7_Optimized_Access := 'TRUE' }
VERSION : 0.1
   VAR_INPUT
      Start : Bool;
      Stop : Bool;
   END_VAR
   VAR_OUTPUT
      Done : Bool;
   END_VAR
   VAR
      "Step" : Int;
      Temp : Array[0..10] of Bool;
      MC_Home_Instance : MC_Home;
      MC_Home_Instance_1 : MC_Home;
      CTRL_HSC_0_Instance : CTRL_HSC;
      IEC_Timer_0_Instance : TON_TIME;
      MC_ReadParam_Instance : MC_ReadParam;
      MC_MoveAbsolute_Instance : MC_MoveAbsolute;
      MC_ReadParam_Instance_1 : MC_ReadParam;
      MC_MoveAbsolute_Instance_1 : MC_MoveAbsolute;
      IEC_Timer_0_Instance_1 : TON_TIME;
      IEC_Timer_0_Instance_2 : TON_TIME;
      IEC_Timer_0_Instance_3 : TON_TIME;
      CTRL_HSC_0_Instance_1 : CTRL_HSC;
      IEC_Timer_0_Instance_4 : TON_TIME;
      IEC_Timer_0_Instance_5 : TON_TIME;
      IEC_Timer_0_Instance_6 : TON_TIME;
   END_VAR
   VAR_TEMP   // added for the SCL form of the ladder/FBD networks
      _w1 : Bool;
      _w2 : Bool;
      _w3 : Bool;
   END_VAR
BEGIN

REGION Network 1
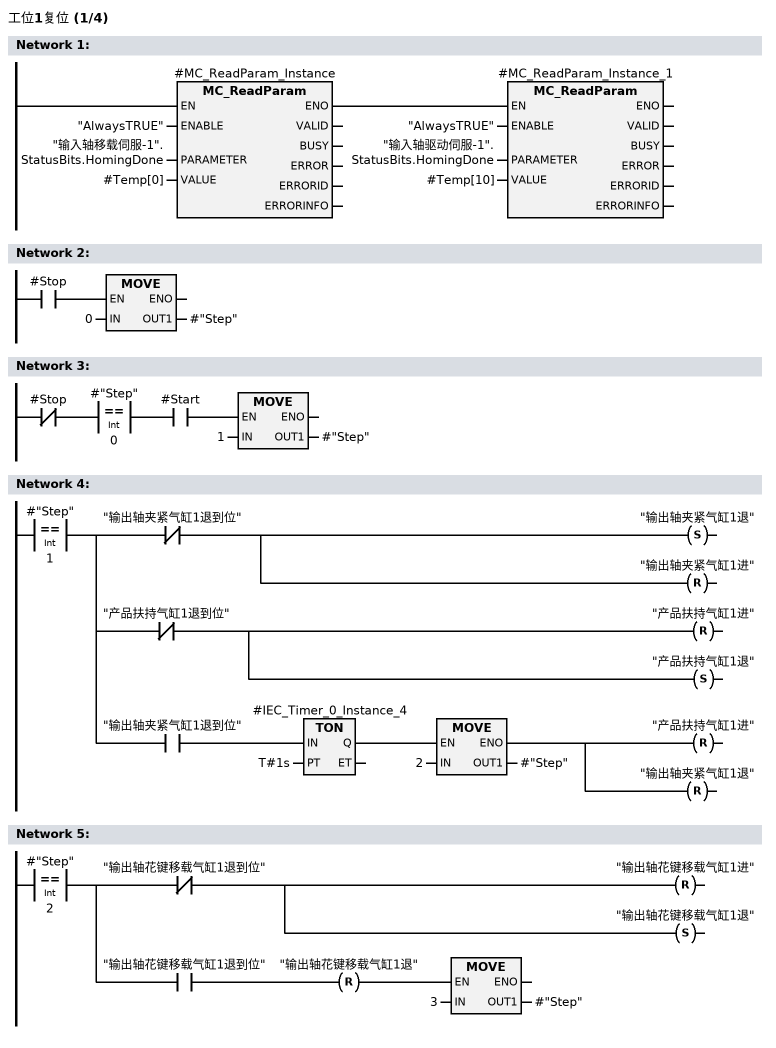
   // ENO of a box is taken as its EN; it also drops when the box reports an error
   #MC_ReadParam_Instance(Enable := "AlwaysTRUE",   // MC_ReadParam
                          Parameter := "输入轴移载伺服-1".StatusBits.HomingDone,
                          Value := #Temp[0]);
   #MC_ReadParam_Instance_1(Enable := "AlwaysTRUE",   // MC_ReadParam
                           Parameter := "输入轴驱动伺服-1".StatusBits.HomingDone,
                           Value := #Temp[10]);
END_REGION

REGION Network 2
   RUNG wire#powerrail
      Contact( #Stop )
      Move(in := 0, out1 => #"Step")
   END_RUNG
   // the same network as SCL:
   IF #Stop THEN #"Step" := 0; END_IF;
END_REGION

REGION Network 3
   RUNG wire#powerrail
      I_Contact( #Stop )
      { S7_Templates := "SrcType := Int" } EQ_Contact(in1 := #"Step", in2 := 0)
      Contact( #Start )
      Move(in := 1, out1 => #"Step")
   END_RUNG
   // the same network as SCL:
   IF NOT #Stop AND (#"Step" = 0) AND #Start THEN #"Step" := 1; END_IF;
END_REGION

REGION Network 4
   #_w1 := #"Step" = 1;
   IF #_w1 AND NOT "输出轴夹紧气缸1退到位" THEN
       "输出轴夹紧气缸1退" := TRUE;
       "输出轴夹紧气缸1进" := FALSE;
   END_IF;
   IF #_w1 AND NOT "产品扶持气缸1退到位" THEN
       "产品扶持气缸1进" := FALSE;
       "产品扶持气缸1退" := TRUE;
   END_IF;
   #IEC_Timer_0_Instance_4(IN := #_w1 AND "输出轴夹紧气缸1退到位", PT := T#1s);   // TON
   IF #IEC_Timer_0_Instance_4.Q THEN
       #"Step" := 2;
       "产品扶持气缸1进" := FALSE;
       "输出轴夹紧气缸1退" := FALSE;
   END_IF;
END_REGION

REGION Network 5
   RUNG wire#powerrail
      { S7_Templates := "SrcType := Int" } EQ_Contact(in1 := #"Step", in2 := 2)
      wire#w1
      I_Contact( "输出轴花键移载气缸1退到位" )
      wire#w2
      R_Coil( "输出轴花键移载气缸1进" )
   END_RUNG
   RUNG wire#w2
      S_Coil( "输出轴花键移载气缸1退" )
   END_RUNG
   RUNG wire#w1
      Contact( "输出轴花键移载气缸1退到位" )
      R_Coil( "输出轴花键移载气缸1退" )
      Move(in := 3, out1 => #"Step")
   END_RUNG
   // the same network as SCL:
   #_w1 := #"Step" = 2;
   IF #_w1 AND NOT "输出轴花键移载气缸1退到位" THEN
       "输出轴花键移载气缸1进" := FALSE;
       "输出轴花键移载气缸1退" := TRUE;
   END_IF;
   IF #_w1 AND "输出轴花键移载气缸1退到位" THEN
       "输出轴花键移载气缸1退" := FALSE;
       #"Step" := 3;
   END_IF;
END_REGION

REGION Network 6
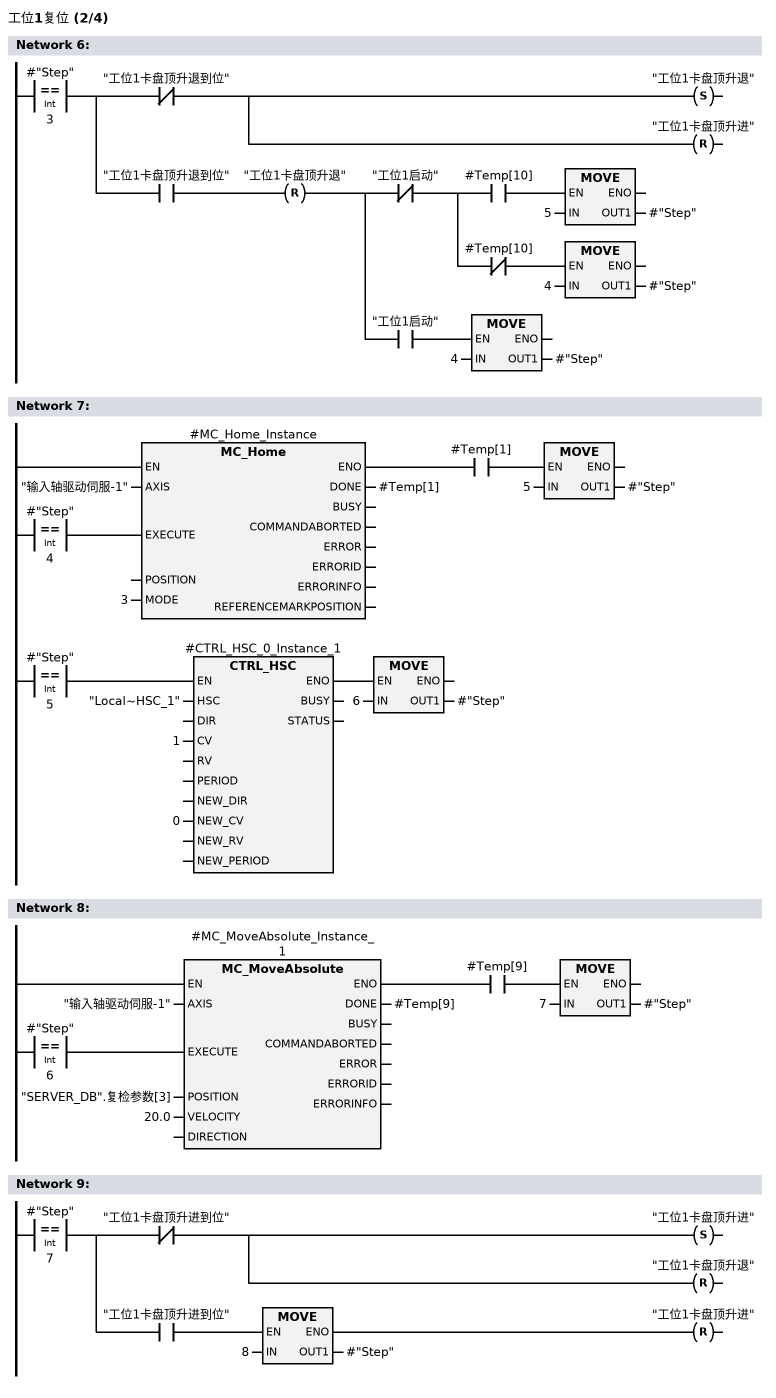
   RUNG wire#powerrail
      { S7_Templates := "SrcType := Int" } EQ_Contact(in1 := #"Step", in2 := 3)
      wire#w1
      I_Contact( "工位1卡盘顶升退到位" )
      wire#w2
      S_Coil( "工位1卡盘顶升退" )
   END_RUNG
   RUNG wire#w2
      R_Coil( "工位1卡盘顶升进" )
   END_RUNG
   RUNG wire#w1
      Contact( "工位1卡盘顶升退到位" )
      R_Coil( "工位1卡盘顶升退" )
      wire#w3
      I_Contact( "工位1启动" )
      wire#w4
      Contact( #Temp[10] )
      Move(in := 5, out1 => #"Step")
   END_RUNG
   RUNG wire#w4
      I_Contact( #Temp[10] )
      Move(in := 4, out1 => #"Step")
   END_RUNG
   RUNG wire#w3
      Contact( "工位1启动" )
      Move(in := 4, out1 => #"Step")
   END_RUNG
   // the same network as SCL:
   #_w1 := #"Step" = 3;
   IF #_w1 AND NOT "工位1卡盘顶升退到位" THEN
       "工位1卡盘顶升退" := TRUE;
       "工位1卡盘顶升进" := FALSE;
   END_IF;
   #_w2 := #_w1 AND "工位1卡盘顶升退到位";
   IF #_w2 THEN "工位1卡盘顶升退" := FALSE; END_IF;
   #_w3 := #_w2 AND NOT "工位1启动";
   IF #_w3 AND #Temp[10] THEN #"Step" := 5; END_IF;
   IF #_w3 AND NOT #Temp[10] THEN #"Step" := 4; END_IF;
   IF #_w2 AND "工位1启动" THEN #"Step" := 4; END_IF;
END_REGION

REGION Network 7
   // ENO of a box is taken as its EN; it also drops when the box reports an error
   #MC_Home_Instance(Axis := "输入轴驱动伺服-1", Execute := #"Step" = 4, Mode := 3, Done => #Temp[1]);   // MC_Home
   IF #Temp[1] THEN #"Step" := 5; END_IF;
   IF #"Step" = 5 THEN
       #CTRL_HSC_0_Instance_1(HSC := "Local~HSC_1", CV := 1, NEW_CV := 0);   // CTRL_HSC
       #"Step" := 6;
   END_IF;
END_REGION

REGION Network 8
   // ENO of a box is taken as its EN; it also drops when the box reports an error
   #MC_MoveAbsolute_Instance_1(Axis := "输入轴驱动伺服-1",   // MC_MoveAbsolute
                           Execute := #"Step" = 6,
                           Position := "SERVER_DB".复检参数[3],
                           Velocity := 20.0,
                           Done => #Temp[9]);
   IF #Temp[9] THEN #"Step" := 7; END_IF;
END_REGION

REGION Network 9
   RUNG wire#powerrail
      { S7_Templates := "SrcType := Int" } EQ_Contact(in1 := #"Step", in2 := 7)
      wire#w1
      I_Contact( "工位1卡盘顶升进到位" )
      wire#w2
      S_Coil( "工位1卡盘顶升进" )
   END_RUNG
   RUNG wire#w2
      R_Coil( "工位1卡盘顶升退" )
   END_RUNG
   RUNG wire#w1
      Contact( "工位1卡盘顶升进到位" )
      Move(in := 8, out1 => #"Step")
      R_Coil( "工位1卡盘顶升进" )
   END_RUNG
   // the same network as SCL:
   #_w1 := #"Step" = 7;
   IF #_w1 AND NOT "工位1卡盘顶升进到位" THEN
       "工位1卡盘顶升进" := TRUE;
       "工位1卡盘顶升退" := FALSE;
   END_IF;
   IF #_w1 AND "工位1卡盘顶升进到位" THEN
       #"Step" := 8;
       "工位1卡盘顶升进" := FALSE;
   END_IF;
END_REGION

REGION Network 10
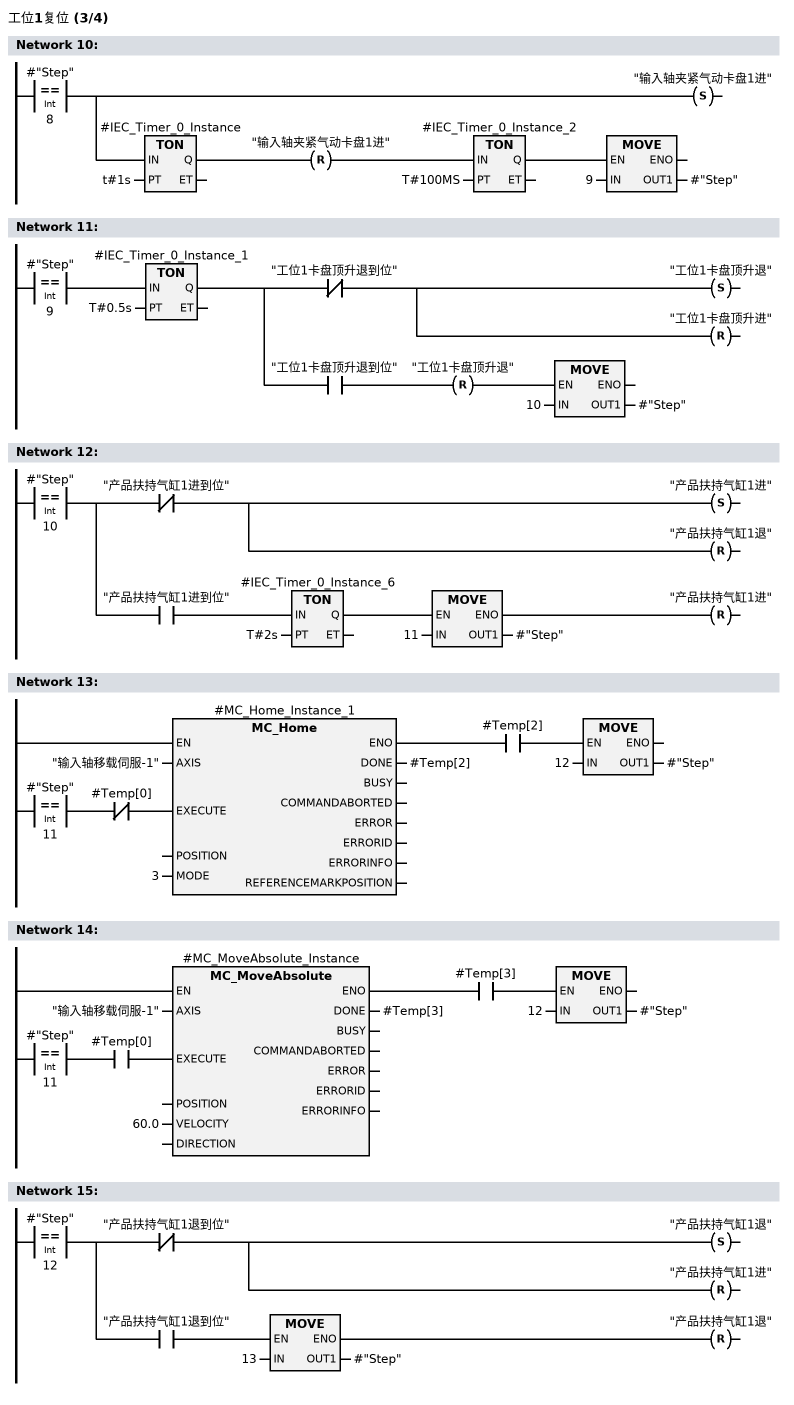
   #_w1 := #"Step" = 8;
   IF #_w1 THEN "输入轴夹紧气动卡盘1进" := TRUE; END_IF;
   #IEC_Timer_0_Instance(IN := #_w1, PT := t#1s);   // TON
   IF #IEC_Timer_0_Instance.Q THEN "输入轴夹紧气动卡盘1进" := FALSE; END_IF;
   #IEC_Timer_0_Instance_2(IN := #IEC_Timer_0_Instance.Q, PT := T#100MS);   // TON
   IF #IEC_Timer_0_Instance_2.Q THEN #"Step" := 9; END_IF;
END_REGION

REGION Network 11
   #IEC_Timer_0_Instance_1(IN := #"Step" = 9, PT := T#0.5s);   // TON
   IF #IEC_Timer_0_Instance_1.Q AND NOT "工位1卡盘顶升退到位" THEN
       "工位1卡盘顶升退" := TRUE;
       "工位1卡盘顶升进" := FALSE;
   END_IF;
   IF #IEC_Timer_0_Instance_1.Q AND "工位1卡盘顶升退到位" THEN
       "工位1卡盘顶升退" := FALSE;
       #"Step" := 10;
   END_IF;
END_REGION

REGION Network 12
   #_w1 := #"Step" = 10;
   IF #_w1 AND NOT "产品扶持气缸1进到位" THEN
       "产品扶持气缸1进" := TRUE;
       "产品扶持气缸1退" := FALSE;
   END_IF;
   #IEC_Timer_0_Instance_6(IN := #_w1 AND "产品扶持气缸1进到位", PT := T#2s);   // TON
   IF #IEC_Timer_0_Instance_6.Q THEN
       #"Step" := 11;
       "产品扶持气缸1进" := FALSE;
   END_IF;
END_REGION

REGION Network 13
   // ENO of a box is taken as its EN; it also drops when the box reports an error
   #MC_Home_Instance_1(Axis := "输入轴移载伺服-1",   // MC_Home
                       Execute := (#"Step" = 11) AND NOT #Temp[0],
                       Mode := 3,
                       Done => #Temp[2]);
   IF #Temp[2] THEN #"Step" := 12; END_IF;
END_REGION

REGION Network 14
   // ENO of a box is taken as its EN; it also drops when the box reports an error
   #MC_MoveAbsolute_Instance(Axis := "输入轴移载伺服-1",   // MC_MoveAbsolute
                           Execute := (#"Step" = 11) AND #Temp[0],
                           Velocity := 60.0,
                           Done => #Temp[3]);
   IF #Temp[3] THEN #"Step" := 12; END_IF;
END_REGION

REGION Network 15
   RUNG wire#powerrail
      { S7_Templates := "SrcType := Int" } EQ_Contact(in1 := #"Step", in2 := 12)
      wire#w1
      I_Contact( "产品扶持气缸1退到位" )
      wire#w2
      S_Coil( "产品扶持气缸1退" )
   END_RUNG
   RUNG wire#w2
      R_Coil( "产品扶持气缸1进" )
   END_RUNG
   RUNG wire#w1
      Contact( "产品扶持气缸1退到位" )
      Move(in := 13, out1 => #"Step")
      R_Coil( "产品扶持气缸1退" )
   END_RUNG
   // the same network as SCL:
   #_w1 := #"Step" = 12;
   IF #_w1 AND NOT "产品扶持气缸1退到位" THEN
       "产品扶持气缸1退" := TRUE;
       "产品扶持气缸1进" := FALSE;
   END_IF;
   IF #_w1 AND "产品扶持气缸1退到位" THEN
       #"Step" := 13;
       "产品扶持气缸1退" := FALSE;
   END_IF;
END_REGION

REGION Network 16
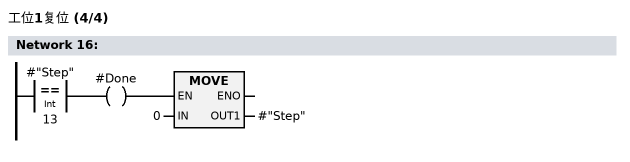
   RUNG wire#powerrail
      { S7_Templates := "SrcType := Int" } EQ_Contact(in1 := #"Step", in2 := 13)
      Coil( #Done )
      Move(in := 0, out1 => #"Step")
   END_RUNG
   // the same network as SCL:
   #Done := #"Step" = 13;
   IF #Done THEN #"Step" := 0; END_IF;
END_REGION
END_FUNCTION_BLOCK

FUNCTION_BLOCK "Alarm"   // FB7, LAD
{ S7_Optimized_Access := 'TRUE' }
VERSION : 0.1
   VAR
      "Step" : Int;
      Temp : Array[0..3] of Bool;
      Error_id : Word;
      IEC_Timer_0_Instance : TON_TIME;
      IEC_Timer_0_Instance_1 : TON_TIME;
      IEC_Timer_0_Instance_2 : TON_TIME;
      IEC_Timer_0_Instance_3 : TON_TIME;
      IEC_Timer_0_Instance_4 : TON_TIME;
      IEC_Timer_0_Instance_5 : TON_TIME;
      IEC_Timer_0_Instance_6 : TON_TIME;
      IEC_Timer_0_Instance_7 : TON_TIME;
      IEC_Timer_0_Instance_8 : TON_TIME;
      IEC_Timer_0_Instance_9 : TON_TIME;
      IEC_Timer_0_Instance_10 : TON_TIME;
   END_VAR
   VAR CONSTANT
      "Time" : Time := T#5000ms;
   END_VAR
   VAR_TEMP   // added for the SCL form of the ladder/FBD networks
      _w1 : Bool;
      _w2 : Bool;
      _w3 : Bool;
      _w4 : Bool;
      _w5 : Bool;
      _w6 : Bool;
      _w7 : Bool;
      _w8 : Bool;
      _w9 : Bool;
      _w10 : Bool;
      _w11 : Bool;
      _w12 : Bool;
   END_VAR
BEGIN

REGION Network 1
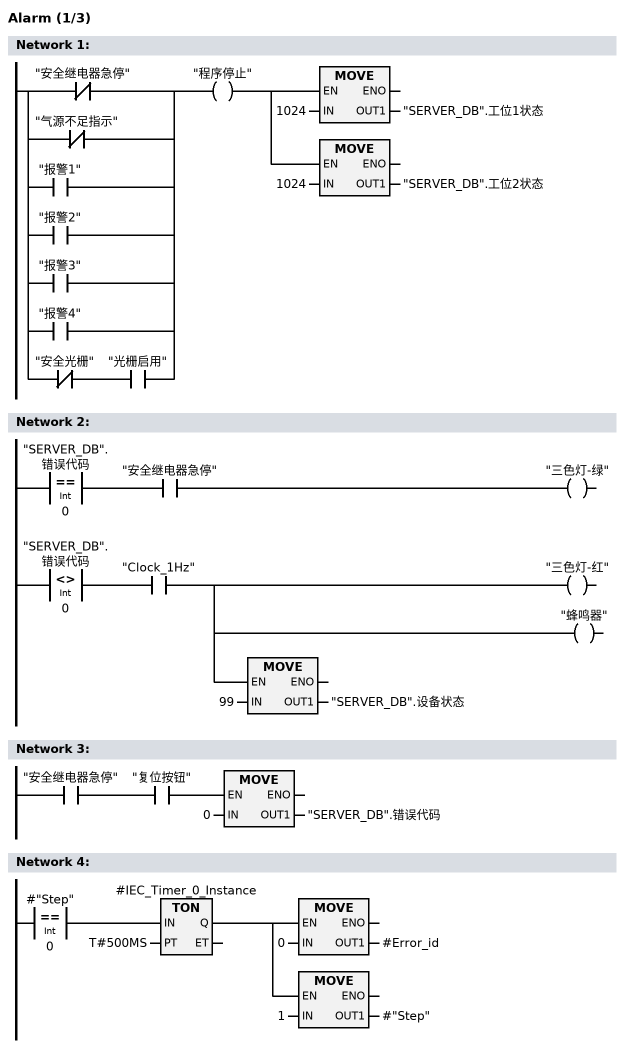
   RUNG wire#powerrail
      I_Contact( "安全继电器急停" )
      wire#w1
      Coil( "程序停止" )
      wire#w2
      Move(in := 1024, out1 => "SERVER_DB".工位1状态)
   END_RUNG
   RUNG wire#powerrail
      I_Contact( "气源不足指示" )
   END_RUNG wire#w1
   RUNG wire#powerrail
      Contact( "报警1" )
   END_RUNG wire#w1
   RUNG wire#powerrail
      Contact( "报警2" )
   END_RUNG wire#w1
   RUNG wire#powerrail
      Contact( "报警3" )
   END_RUNG wire#w1
   RUNG wire#powerrail
      Contact( "报警4" )
   END_RUNG wire#w1
   RUNG wire#powerrail
      I_Contact( "安全光栅" )
      Contact( "光栅启用" )
   END_RUNG wire#w1
   RUNG wire#w2
      Move(in := 1024, out1 => "SERVER_DB".工位2状态)
   END_RUNG
   // the same network as SCL:
   "程序停止" := NOT "安全继电器急停" OR NOT "气源不足指示" OR "报警1" OR "报警2" OR "报警3" OR "报警4" OR (NOT "安全光栅" AND "光栅启用");
   IF "程序停止" THEN
       "SERVER_DB".工位1状态 := 1024;
       "SERVER_DB".工位2状态 := 1024;
   END_IF;
END_REGION

REGION Network 2
   RUNG wire#powerrail
      { S7_Templates := "SrcType := Int" } EQ_Contact(in1 := "SERVER_DB".错误代码, in2 := 0)
      Contact( "安全继电器急停" )
      Coil( "三色灯-绿" )
   END_RUNG
   RUNG wire#powerrail
      { S7_Templates := "SrcType := Int" } NE_Contact(in1 := "SERVER_DB".错误代码, in2 := 0)
      Contact( "Clock_1Hz" )
      wire#w1
      Coil( "三色灯-红" )
   END_RUNG
   RUNG wire#w1
      Coil( "蜂鸣器" )
   END_RUNG
   RUNG wire#w1
      Move(in := 99, out1 => "SERVER_DB".设备状态)
   END_RUNG
   // the same network as SCL:
   "三色灯-绿" := ("SERVER_DB".错误代码 = 0) AND "安全继电器急停";
   "三色灯-红" := ("SERVER_DB".错误代码 <> 0) AND "Clock_1Hz";
   "蜂鸣器" := "三色灯-红";
   IF "三色灯-红" THEN "SERVER_DB".设备状态 := 99; END_IF;
END_REGION

REGION Network 3
   RUNG wire#powerrail
      Contact( "安全继电器急停" )
      Contact( "复位按钮" )
      Move(in := 0, out1 => "SERVER_DB".错误代码)
   END_RUNG
   // the same network as SCL:
   IF "安全继电器急停" AND "复位按钮" THEN "SERVER_DB".错误代码 := 0; END_IF;
END_REGION

REGION Network 4
   #IEC_Timer_0_Instance(IN := #"Step" = 0, PT := T#500MS);   // TON
   IF #IEC_Timer_0_Instance.Q THEN
       #Error_id := 0;
       #"Step" := 1;
   END_IF;
END_REGION

REGION Network 5
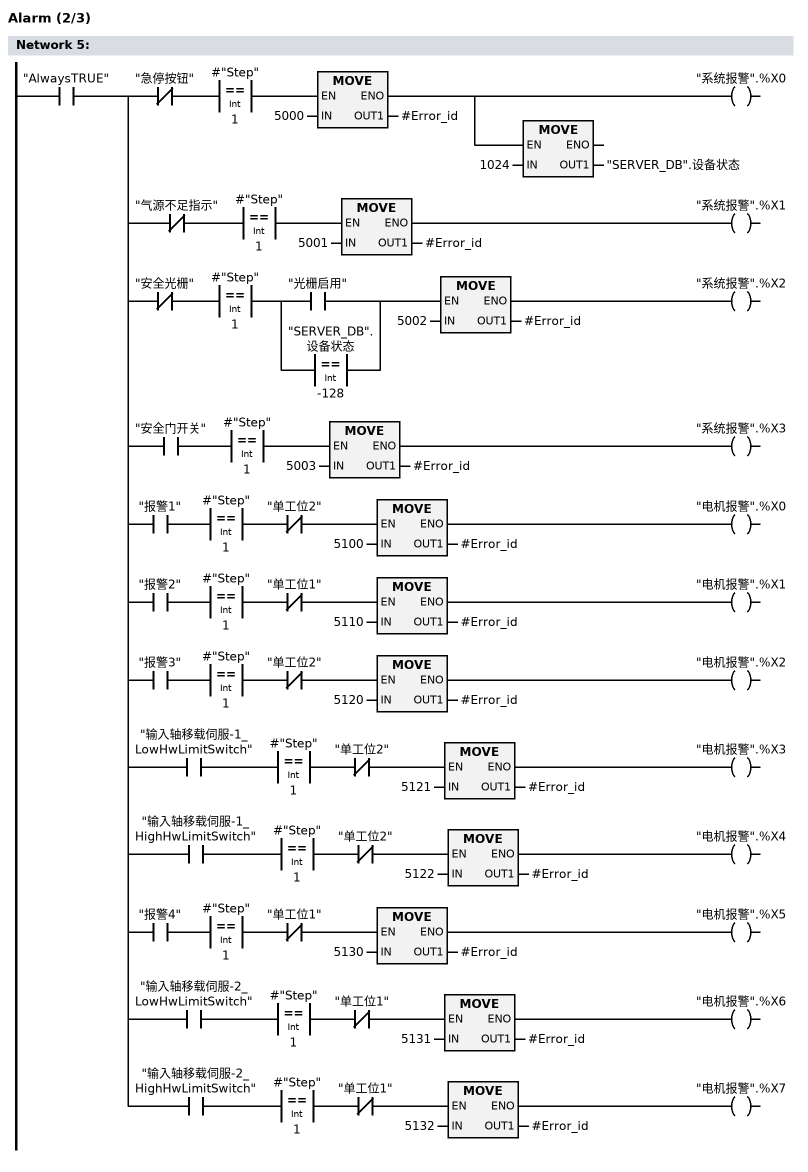
   RUNG wire#powerrail
      Contact( "AlwaysTRUE" )
      wire#w1
      I_Contact( "急停按钮" )
      { S7_Templates := "SrcType := Int" } EQ_Contact(in1 := #"Step", in2 := 1)
      Move(in := 5000, out1 => #Error_id)
      wire#w2
      Coil( "系统报警".%X0 )
   END_RUNG
   RUNG wire#w2
      Move(in := 1024, out1 => "SERVER_DB".设备状态)
   END_RUNG
   RUNG wire#w1
      I_Contact( "气源不足指示" )
      { S7_Templates := "SrcType := Int" } EQ_Contact(in1 := #"Step", in2 := 1)
      Move(in := 5001, out1 => #Error_id)
      Coil( "系统报警".%X1 )
   END_RUNG
   RUNG wire#w1
      I_Contact( "安全光栅" )
      { S7_Templates := "SrcType := Int" } EQ_Contact(in1 := #"Step", in2 := 1)
      wire#w3
      Contact( "光栅启用" )
      wire#w4
      Move(in := 5002, out1 => #Error_id)
      Coil( "系统报警".%X2 )
   END_RUNG
   RUNG wire#w3
      { S7_Templates := "SrcType := Int" } EQ_Contact(in1 := "SERVER_DB".设备状态, in2 := -128)
   END_RUNG wire#w4
   RUNG wire#w1
      Contact( "安全门开关" )
      { S7_Templates := "SrcType := Int" } EQ_Contact(in1 := #"Step", in2 := 1)
      Move(in := 5003, out1 => #Error_id)
      Coil( "系统报警".%X3 )
   END_RUNG
   RUNG wire#w1
      Contact( "报警1" )
      { S7_Templates := "SrcType := Int" } EQ_Contact(in1 := #"Step", in2 := 1)
      I_Contact( "单工位2" )
      Move(in := 5100, out1 => #Error_id)
      Coil( "电机报警".%X0 )
   END_RUNG
   RUNG wire#w1
      Contact( "报警2" )
      { S7_Templates := "SrcType := Int" } EQ_Contact(in1 := #"Step", in2 := 1)
      I_Contact( "单工位1" )
      Move(in := 5110, out1 => #Error_id)
      Coil( "电机报警".%X1 )
   END_RUNG
   RUNG wire#w1
      Contact( "报警3" )
      { S7_Templates := "SrcType := Int" } EQ_Contact(in1 := #"Step", in2 := 1)
      I_Contact( "单工位2" )
      Move(in := 5120, out1 => #Error_id)
      Coil( "电机报警".%X2 )
   END_RUNG
   RUNG wire#w1
      Contact( "输入轴移载伺服-1_LowHwLimitSwitch" )
      { S7_Templates := "SrcType := Int" } EQ_Contact(in1 := #"Step", in2 := 1)
      I_Contact( "单工位2" )
      Move(in := 5121, out1 => #Error_id)
      Coil( "电机报警".%X3 )
   END_RUNG
   RUNG wire#w1
      Contact( "输入轴移载伺服-1_HighHwLimitSwitch" )
      { S7_Templates := "SrcType := Int" } EQ_Contact(in1 := #"Step", in2 := 1)
      I_Contact( "单工位2" )
      Move(in := 5122, out1 => #Error_id)
      Coil( "电机报警".%X4 )
   END_RUNG
   RUNG wire#w1
      Contact( "报警4" )
      { S7_Templates := "SrcType := Int" } EQ_Contact(in1 := #"Step", in2 := 1)
      I_Contact( "单工位1" )
      Move(in := 5130, out1 => #Error_id)
      Coil( "电机报警".%X5 )
   END_RUNG
   RUNG wire#w1
      Contact( "输入轴移载伺服-2_LowHwLimitSwitch" )
      { S7_Templates := "SrcType := Int" } EQ_Contact(in1 := #"Step", in2 := 1)
      I_Contact( "单工位1" )
      Move(in := 5131, out1 => #Error_id)
      Coil( "电机报警".%X6 )
   END_RUNG
   RUNG wire#w1
      Contact( "输入轴移载伺服-2_HighHwLimitSwitch" )
      { S7_Templates := "SrcType := Int" } EQ_Contact(in1 := #"Step", in2 := 1)
      I_Contact( "单工位1" )
      Move(in := 5132, out1 => #Error_id)
      Coil( "电机报警".%X7 )
   END_RUNG
   // the same network as SCL:
   #_w1 := "AlwaysTRUE" AND NOT "急停按钮" AND (#"Step" = 1);
   IF #_w1 THEN #Error_id := 5000; END_IF;
   "系统报警".%X0 := #_w1;
   IF #_w1 THEN "SERVER_DB".设备状态 := 1024; END_IF;
   #_w2 := "AlwaysTRUE" AND NOT "气源不足指示" AND (#"Step" = 1);
   IF #_w2 THEN #Error_id := 5001; END_IF;
   "系统报警".%X1 := #_w2;
   #_w3 := "AlwaysTRUE" AND NOT "安全光栅" AND (#"Step" = 1) AND ("光栅启用" OR ("SERVER_DB".设备状态 = (-128)));
   IF #_w3 THEN #Error_id := 5002; END_IF;
   "系统报警".%X2 := #_w3;
   #_w4 := "AlwaysTRUE" AND "安全门开关" AND (#"Step" = 1);
   IF #_w4 THEN #Error_id := 5003; END_IF;
   "系统报警".%X3 := #_w4;
   #_w5 := "AlwaysTRUE" AND "报警1" AND (#"Step" = 1) AND NOT "单工位2";
   IF #_w5 THEN #Error_id := 5100; END_IF;
   "电机报警".%X0 := #_w5;
   #_w6 := "AlwaysTRUE" AND "报警2" AND (#"Step" = 1) AND NOT "单工位1";
   IF #_w6 THEN #Error_id := 5110; END_IF;
   "电机报警".%X1 := #_w6;
   #_w7 := "AlwaysTRUE" AND "报警3" AND (#"Step" = 1) AND NOT "单工位2";
   IF #_w7 THEN #Error_id := 5120; END_IF;
   "电机报警".%X2 := #_w7;
   #_w8 := "AlwaysTRUE" AND "输入轴移载伺服-1_LowHwLimitSwitch" AND (#"Step" = 1) AND NOT "单工位2";
   IF #_w8 THEN #Error_id := 5121; END_IF;
   "电机报警".%X3 := #_w8;
   #_w9 := "AlwaysTRUE" AND "输入轴移载伺服-1_HighHwLimitSwitch" AND (#"Step" = 1) AND NOT "单工位2";
   IF #_w9 THEN #Error_id := 5122; END_IF;
   "电机报警".%X4 := #_w9;
   #_w10 := "AlwaysTRUE" AND "报警4" AND (#"Step" = 1) AND NOT "单工位1";
   IF #_w10 THEN #Error_id := 5130; END_IF;
   "电机报警".%X5 := #_w10;
   #_w11 := "AlwaysTRUE" AND "输入轴移载伺服-2_LowHwLimitSwitch" AND (#"Step" = 1) AND NOT "单工位1";
   IF #_w11 THEN #Error_id := 5131; END_IF;
   "电机报警".%X6 := #_w11;
   #_w12 := "AlwaysTRUE" AND "输入轴移载伺服-2_HighHwLimitSwitch" AND (#"Step" = 1) AND NOT "单工位1";
   IF #_w12 THEN #Error_id := 5132; END_IF;
   "电机报警".%X7 := #_w12;
END_REGION

REGION Network 6
   // 到位故障
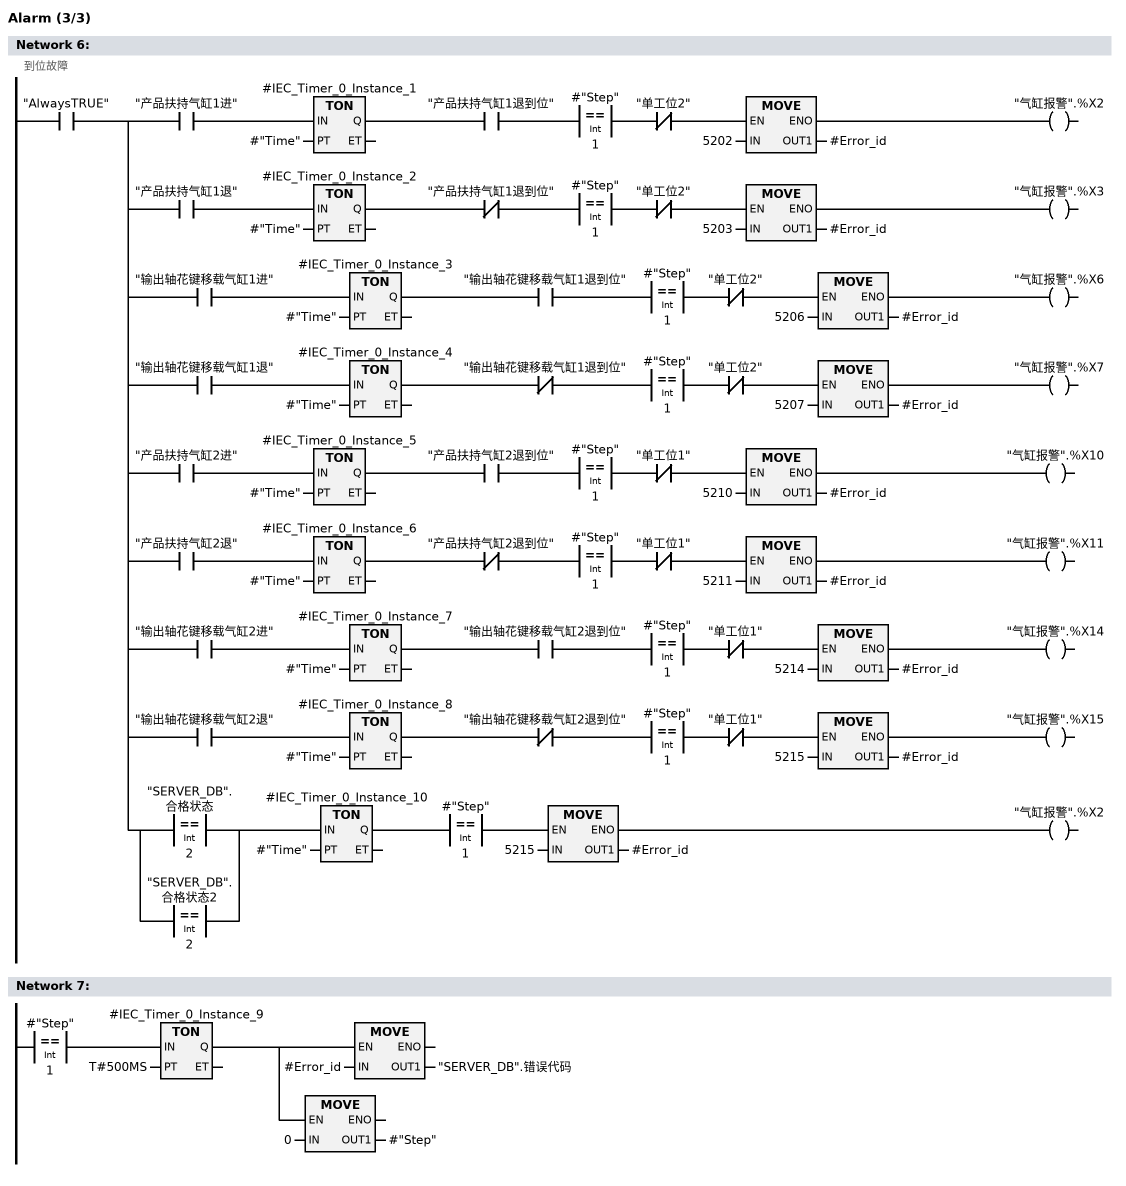
   #IEC_Timer_0_Instance_1(IN := "AlwaysTRUE" AND "产品扶持气缸1进", PT := #"Time");   // TON
   #_w1 := #IEC_Timer_0_Instance_1.Q AND "产品扶持气缸1退到位" AND (#"Step" = 1) AND NOT "单工位2";
   IF #_w1 THEN #Error_id := 5202; END_IF;
   "气缸报警".%X2 := #_w1;
   #IEC_Timer_0_Instance_2(IN := "AlwaysTRUE" AND "产品扶持气缸1退", PT := #"Time");   // TON
   #_w2 := #IEC_Timer_0_Instance_2.Q AND NOT "产品扶持气缸1退到位" AND (#"Step" = 1) AND NOT "单工位2";
   IF #_w2 THEN #Error_id := 5203; END_IF;
   "气缸报警".%X3 := #_w2;
   #IEC_Timer_0_Instance_3(IN := "AlwaysTRUE" AND "输出轴花键移载气缸1进", PT := #"Time");   // TON
   #_w3 := #IEC_Timer_0_Instance_3.Q AND "输出轴花键移载气缸1退到位" AND (#"Step" = 1) AND NOT "单工位2";
   IF #_w3 THEN #Error_id := 5206; END_IF;
   "气缸报警".%X6 := #_w3;
   #IEC_Timer_0_Instance_4(IN := "AlwaysTRUE" AND "输出轴花键移载气缸1退", PT := #"Time");   // TON
   #_w4 := #IEC_Timer_0_Instance_4.Q AND NOT "输出轴花键移载气缸1退到位" AND (#"Step" = 1) AND NOT "单工位2";
   IF #_w4 THEN #Error_id := 5207; END_IF;
   "气缸报警".%X7 := #_w4;
   #IEC_Timer_0_Instance_5(IN := "AlwaysTRUE" AND "产品扶持气缸2进", PT := #"Time");   // TON
   #_w5 := #IEC_Timer_0_Instance_5.Q AND "产品扶持气缸2退到位" AND (#"Step" = 1) AND NOT "单工位1";
   IF #_w5 THEN #Error_id := 5210; END_IF;
   "气缸报警".%X10 := #_w5;
   #IEC_Timer_0_Instance_6(IN := "AlwaysTRUE" AND "产品扶持气缸2退", PT := #"Time");   // TON
   #_w6 := #IEC_Timer_0_Instance_6.Q AND NOT "产品扶持气缸2退到位" AND (#"Step" = 1) AND NOT "单工位1";
   IF #_w6 THEN #Error_id := 5211; END_IF;
   "气缸报警".%X11 := #_w6;
   #IEC_Timer_0_Instance_7(IN := "AlwaysTRUE" AND "输出轴花键移载气缸2进", PT := #"Time");   // TON
   #_w7 := #IEC_Timer_0_Instance_7.Q AND "输出轴花键移载气缸2退到位" AND (#"Step" = 1) AND NOT "单工位1";
   IF #_w7 THEN #Error_id := 5214; END_IF;
   "气缸报警".%X14 := #_w7;
   #IEC_Timer_0_Instance_8(IN := "AlwaysTRUE" AND "输出轴花键移载气缸2退", PT := #"Time");   // TON
   #_w8 := #IEC_Timer_0_Instance_8.Q AND NOT "输出轴花键移载气缸2退到位" AND (#"Step" = 1) AND NOT "单工位1";
   IF #_w8 THEN #Error_id := 5215; END_IF;
   "气缸报警".%X15 := #_w8;
   #IEC_Timer_0_Instance_10(IN := "AlwaysTRUE" AND (("SERVER_DB".合格状态 = 2) OR ("SERVER_DB".合格状态2 = 2)),   // TON
                           PT := #"Time");
   #_w9 := #IEC_Timer_0_Instance_10.Q AND (#"Step" = 1);
   IF #_w9 THEN #Error_id := 5215; END_IF;
   "气缸报警".%X2 := #_w9;
END_REGION

REGION Network 7
   #IEC_Timer_0_Instance_9(IN := #"Step" = 1, PT := T#500MS);   // TON
   IF #IEC_Timer_0_Instance_9.Q THEN
       "SERVER_DB".错误代码 := #Error_id;
       #"Step" := 0;
   END_IF;
END_REGION
END_FUNCTION_BLOCK

FUNCTION_BLOCK "工位2复位"   // FB8, LAD
{ S7_Optimized_Access := 'TRUE' }
VERSION : 0.1
   VAR_INPUT
      Start : Bool;
      Stop : Bool;
   END_VAR
   VAR_OUTPUT
      Done : Bool;
   END_VAR
   VAR
      "Step" : Int;
      Temp : Array[0..10] of Bool;
      MC_Home_Instance : MC_Home;
      MC_Home_Instance_1 : MC_Home;
      CTRL_HSC_0_Instance : CTRL_HSC;
      IEC_Timer_0_Instance : TON_TIME;
      MC_ReadParam_Instance : MC_ReadParam;
      MC_MoveAbsolute_Instance : MC_MoveAbsolute;
      MC_ReadParam_Instance_1 : MC_ReadParam;
      MC_MoveAbsolute_Instance_1 : MC_MoveAbsolute;
      IEC_Timer_0_Instance_1 : TON_TIME;
      IEC_Timer_0_Instance_2 : TON_TIME;
      IEC_Timer_0_Instance_3 : TON_TIME;
      CTRL_HSC_0_Instance_1 : CTRL_HSC;
      IEC_Timer_0_Instance_4 : TON_TIME;
      IEC_Timer_0_Instance_5 : TON_TIME;
      IEC_Timer_0_Instance_6 : TON_TIME;
   END_VAR
   VAR_TEMP   // added for the SCL form of the ladder/FBD networks
      _w1 : Bool;
      _w2 : Bool;
      _w3 : Bool;
   END_VAR
BEGIN

REGION Network 1
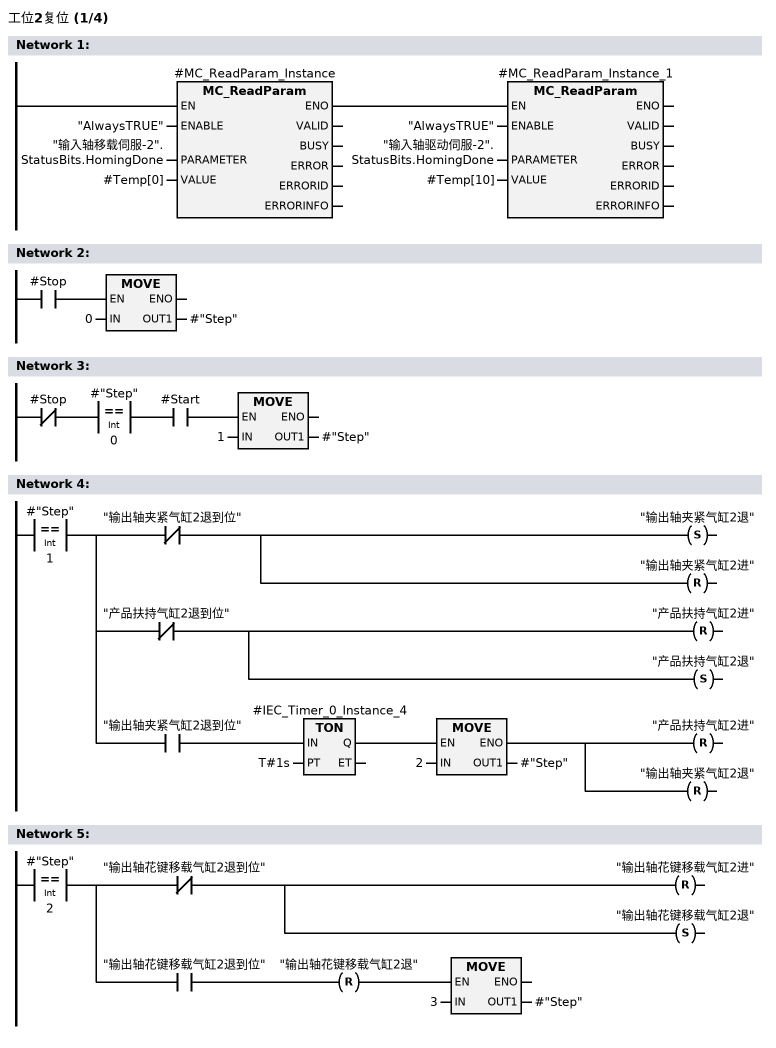
   // ENO of a box is taken as its EN; it also drops when the box reports an error
   #MC_ReadParam_Instance(Enable := "AlwaysTRUE",   // MC_ReadParam
                          Parameter := "输入轴移载伺服-2".StatusBits.HomingDone,
                          Value := #Temp[0]);
   #MC_ReadParam_Instance_1(Enable := "AlwaysTRUE",   // MC_ReadParam
                           Parameter := "输入轴驱动伺服-2".StatusBits.HomingDone,
                           Value := #Temp[10]);
END_REGION

REGION Network 2
   RUNG wire#powerrail
      Contact( #Stop )
      Move(in := 0, out1 => #"Step")
   END_RUNG
   // the same network as SCL:
   IF #Stop THEN #"Step" := 0; END_IF;
END_REGION

REGION Network 3
   RUNG wire#powerrail
      I_Contact( #Stop )
      { S7_Templates := "SrcType := Int" } EQ_Contact(in1 := #"Step", in2 := 0)
      Contact( #Start )
      Move(in := 1, out1 => #"Step")
   END_RUNG
   // the same network as SCL:
   IF NOT #Stop AND (#"Step" = 0) AND #Start THEN #"Step" := 1; END_IF;
END_REGION

REGION Network 4
   #_w1 := #"Step" = 1;
   IF #_w1 AND NOT "输出轴夹紧气缸2退到位" THEN
       "输出轴夹紧气缸2退" := TRUE;
       "输出轴夹紧气缸2进" := FALSE;
   END_IF;
   IF #_w1 AND NOT "产品扶持气缸2退到位" THEN
       "产品扶持气缸2进" := FALSE;
       "产品扶持气缸2退" := TRUE;
   END_IF;
   #IEC_Timer_0_Instance_4(IN := #_w1 AND "输出轴夹紧气缸2退到位", PT := T#1s);   // TON
   IF #IEC_Timer_0_Instance_4.Q THEN
       #"Step" := 2;
       "产品扶持气缸2进" := FALSE;
       "输出轴夹紧气缸2退" := FALSE;
   END_IF;
END_REGION

REGION Network 5
   RUNG wire#powerrail
      { S7_Templates := "SrcType := Int" } EQ_Contact(in1 := #"Step", in2 := 2)
      wire#w1
      I_Contact( "输出轴花键移载气缸2退到位" )
      wire#w2
      R_Coil( "输出轴花键移载气缸2进" )
   END_RUNG
   RUNG wire#w2
      S_Coil( "输出轴花键移载气缸2退" )
   END_RUNG
   RUNG wire#w1
      Contact( "输出轴花键移载气缸2退到位" )
      R_Coil( "输出轴花键移载气缸2退" )
      Move(in := 3, out1 => #"Step")
   END_RUNG
   // the same network as SCL:
   #_w1 := #"Step" = 2;
   IF #_w1 AND NOT "输出轴花键移载气缸2退到位" THEN
       "输出轴花键移载气缸2进" := FALSE;
       "输出轴花键移载气缸2退" := TRUE;
   END_IF;
   IF #_w1 AND "输出轴花键移载气缸2退到位" THEN
       "输出轴花键移载气缸2退" := FALSE;
       #"Step" := 3;
   END_IF;
END_REGION

REGION Network 6
